(* Logix 5000 project; controller IF2_DEMO Emulate 5570 rev 20.12; software revision 20.04 *)
// RSTechEd 2013 Demo

TASK MainTask (continuous, watchdog 100000 ms) : Main, FillerD, LabelerD
TASK MotionTiming (periodic, rate 25 ms, priority 2, watchdog 50000 ms) : MotionProg

MODULES
   Local : Emulate 5570 (ICP 2, rev 20.12)
END_MODULES

TYPE Controls :   // Workcell Status
STRUCT
   Standby : BOOL;
   StandbyCode : INT;
   Run : BOOL;
   Auto : BOOL;
   Run_sw : BOOL;
END_STRUCT
END_TYPE

TYPE Counts :   // Production Information - Part Counts
STRUCT
   Total : DINT;
   Good : DINT;
   Scrap : DINT;
   BottlesMin : DINT;
END_STRUCT
END_TYPE

TYPE DownTime :   // DownTime Category
STRUCT
   Breakdown : BOOL;
   BreakdownCode : INT;
   UnschedMaint : BOOL;
   Testing : BOOL;
END_STRUCT
END_TYPE

TYPE Event_Triggers :
STRUCT
   EventTrigger : INT;
END_STRUCT
END_TYPE

TYPE Events :
STRUCT
   DownTime : DownTime;
   Operate : Operate;
   Control : Controls;
END_STRUCT
END_TYPE

TYPE FTVPDemoEvents :
STRUCT
   DownTime : DownTime;
   Operate : Operate;
   Control : Controls;
END_STRUCT
END_TYPE

TYPE FTVPDemoLine :
STRUCT
   Downtime : DINT;   // Line Downtime Value
   Runstate : BOOL;   // Running status of the line
   OutputTarget : REAL;   // Target value for production output
   OutputActual : REAL;   // Actual Value of Production Output
   Quality : REAL;   // Line Quality Value
   Rejects : REAL;   // Line Reject Count
END_STRUCT
END_TYPE

TYPE FTVPDemoProduct :
STRUCT
   ProductID : STRING;
   Recipe : STRING;
END_STRUCT
END_TYPE

TYPE FTVPDemoWorkCell :
STRUCT
   LineName : STRING;
   RunState : BOOL;
   Temperature : DINT;
   GoodParts : INT;
   ScrapParts : INT;
   ScrapRate : DINT;
   ProductionRate : DINT;
   Pressure : DINT;
   OrderName : STRING;
   CustomerName : STRING;
   PartName : STRING;
END_STRUCT
END_TYPE

TYPE FTVPSampleMaintenance :
STRUCT
   OperatorLog : STRING;
   MaintenanceActual : DINT;
   MaintenancePlanned : DINT;
   ScheduledDownTime : STRING;
END_STRUCT
END_TYPE

TYPE HMIVars :   // Operator Interface Data
STRUCT
   ScrapRate : REAL;
   SpeedControl : REAL;
   PrevSpeed : REAL;
   CurrentProductionRate : REAL;
   PartCountRollOver : DINT;
   MfgTimeBase : INT;
   MaxEventDur : REAL;
   MinEventDur : REAL;
   EventsPerHr : INT;
   EventDur : REAL;
   RunDur : REAL;
   MinRunDur : REAL;
END_STRUCT
END_TYPE

TYPE IF_OEE :
STRUCT
   Quality : REAL;
   Efficiency : REAL;
   AvailableTime : REAL;
END_STRUCT
END_TYPE

TYPE IPTankLevel :
STRUCT
   Water : Level;
   Chemical : Level;
   Sanitizer : Level;
   RecoveredWater : Level;
END_STRUCT
END_TYPE

TYPE Level :
STRUCT
   Minimum : DINT;
   Maximum : DINT;
   Value : DINT;
END_STRUCT
END_TYPE

TYPE LineData :
STRUCT
   CustomerName : STRING[10];
   PartName : STRING[10];
   OrderName : STRING[10];
   OrderQty : DINT;
END_STRUCT
END_TYPE

TYPE MfgOrders :   // Downloaded Manufacturing Order Details
STRUCT
   CustomerName : STRING;
   OrderName : STRING;
   GetNextOrder : BOOL;
   GetNextOrderStatus : INT;
   OrderQty : DINT;
   OrderQtyStart : DINT;
   ProdRate : REAL;
   SetupTime : REAL;
   PartName : STRING;
   WorkcellName : STRING;
   OperationId : DINT;
   PartNameSav : STRING;
END_STRUCT
END_TYPE

TYPE MLHMI :
STRUCT
   HelpInfo : INT;
   Motor1AmpRate : INT;
   Motor1HighTemp : BOOL;
   Motor1Overload : BOOL;
   Motor2AmpRate : INT;
   Motor2HighTemp : BOOL;
   Motor2Overload : BOOL;
   CustomerName : STRING;
   OEE : INT;
   OrderQTY : INT;
   PartName : STRING;
   ProdRate : INT;
   SetUpTime : INT;
   OrderName : STRING;
END_STRUCT
END_TYPE

TYPE MotionVars :   // Operator Interface Data
STRUCT
   Motion : REAL;
   MotionFactor : REAL;
   MotionMax : REAL;
END_STRUCT
END_TYPE

TYPE OEE :   // Operational Equipment Effectiveness
STRUCT
   IdealCycleTime : REAL;
   Parts : Counts;
END_STRUCT
END_TYPE

TYPE Operate :   // Events related to Operating Workcells
STRUCT
   Setup : BOOL;
   Load : BOOL;
   OrderProc : BOOL;
END_STRUCT
END_TYPE

TYPE PFlex700_Input_I0 :
STRUCT
   DriveStatus : INT;
   DriveStatus_Ready : BOOL;
   DriveStatus_Active : BOOL;
   DriveStatus_CommandDir : BOOL;
   DriveStatus_ActualDir : BOOL;
   DriveStatus_Accelerating : BOOL;
   DriveStatus_Decelerating : BOOL;
   DriveStatus_Alarm : BOOL;
   DriveStatus_Faulted : BOOL;
   DriveStatus_AtSpeed : BOOL;
   DriveStatus_LocalID0 : BOOL;
   DriveStatus_LocalID1 : BOOL;
   DriveStatus_LocalID2 : BOOL;
   DriveStatus_SpdRefID0 : BOOL;
   DriveStatus_SpdRefID1 : BOOL;
   DriveStatus_SpdRefID2 : BOOL;
   DriveStatus_SpdRefID3 : BOOL;
   OutputFreq : INT;
   AccelTime1 : INT;
   DecelTime1 : INT;
   Fault1Code : INT;
   DCBusVoltage : INT;
   OutputCurrent : INT;
   Undefined_C2 : INT;
END_STRUCT
END_TYPE

TYPE PFlex700_Output_O0 :
STRUCT
   DriveLogicRslt : INT;
   DriveLogicRslt_Stop : BOOL;
   DriveLogicRslt_Start : BOOL;
   DriveLogicRslt_Jog : BOOL;
   DriveLogicRslt_ClearFault : BOOL;
   DriveLogicRslt_Forward : BOOL;
   DriveLogicRslt_Reverse : BOOL;
   DriveLogicRslt_LocalContrl : BOOL;
   DriveLogicRslt_MOPInc : BOOL;
   DriveLogicRslt_Accel1 : BOOL;
   DriveLogicRslt_Accel2 : BOOL;
   DriveLogicRslt_Decel1 : BOOL;
   DriveLogicRslt_Decel2 : BOOL;
   DriveLogicRslt_SpdRefID0 : BOOL;
   DriveLogicRslt_SpdRefID1 : BOOL;
   DriveLogicRslt_SpdRefID2 : BOOL;
   DriveLogicRslt_MOPDec : BOOL;
   CommandedFreq : INT;
   AccelTime1 : INT;
   DecelTime1 : INT;
   Undefined_B1 : INT;
   Undefined_B2 : INT;
   Undefined_C1 : INT;
   Undefined_C2 : INT;
END_STRUCT
END_TYPE

TYPE Plant :
STRUCT
   Downtime : REAL;
   Output : REAL;
   Quality : REAL;
END_STRUCT
END_TYPE

TYPE SimVars :   // Variables to Simulated Production
STRUCT
   Cycle : TIMER;
   Run : TIMER;
   Event : TIMER;
   Setup : TIMER;
   Good : REAL;
   Scrap : REAL;
   GoToRun : BOOL;
   GoToEvent : BOOL;
   EventNumber : INT;
   UtilityBool : BOOL[32];
END_STRUCT
END_TYPE

TYPE SodaRecipe :
STRUCT
   Water : DINT;
   Syrup : DINT;
   Acid : DINT;
   CarbonDioxide : DINT;
   Flavor : STRING;
END_STRUCT
END_TYPE

TYPE State :
STRUCT
   LineState : STRING;
END_STRUCT
END_TYPE

TYPE Tank :   // Blending Tanks
STRUCT
   Level : DINT;
   Fill_Valve : STRING;   // 0 = Open, 1 = closed
   Discharge_Valve : STRING;   // 0 = Open, 1 = closed
   CIP_Time : STRING;
   Name : STRING;
END_STRUCT
END_TYPE

TYPE WC :
STRUCT
   EventTrigger : DINT[3];
   EventValue_REAL : REAL[46];
   FlexREAL : REAL[6];
   FlexSTRING : STRING[10];
   IdealCT : REAL;   // Ideal Cycle Time
   TotalParts : REAL;   // Total Parts Produced
   GoodParts : REAL;   // Good Parts Produced
   ScrapParts : REAL;   // Scrap Parts Produced
   EventValueSTRING : STRING[5];
   Shift : REAL;   // Shift Value
   MonitorValue : REAL[25];
   PV : REAL[5];
   FlexINT : INT[6];
END_STRUCT
END_TYPE

TYPE WorkOrder :
STRUCT
   CustomerName : STRING;
   PartName : STRING;
   OrderName : STRING;
   OrderNumber : INT;
   OrderQty : INT;
END_STRUCT
END_TYPE

ADD_ON_INSTRUCTION PFlex_700_AOI   (* revision 1.0 031707 *)
VAR_INPUT
   Cmd_OperOperReq : BOOL;
   Cmd_ProgOperReq : BOOL;
END_VAR
VAR_OUTPUT
   Sts_OperatorModeEnabled : BOOL; {access Read Only, visible}
END_VAR
VAR_INPUT
   Cmd_OperProgReq : BOOL;
   Cmd_ProgProgReq : BOOL;
END_VAR
VAR_OUTPUT
   Sts_ProgramModeEnabled : BOOL; {access Read Only, visible}
   Sts_CommFault : BOOL; {access Read Only, visible}
END_VAR
VAR_INPUT
   Cmd_StartOper : BOOL;
   Cmd_StartProg : BOOL;
   Cmd_StopOper : BOOL;
   Cmd_StopProg : BOOL;
   Cmd_ResetOper : BOOL;
   Cmd_ResetProg : BOOL;
   Cmd_JogOper : BOOL;
   Cmd_JogProg : BOOL;
   Cmd_FwdOper : BOOL;
   Cmd_FwdProg : BOOL;
   Cmd_RevOper : BOOL;
   Cmd_RevProg : BOOL;
   Set_SpeedOper : INT;
   Set_SpeedProg : INT;
   Set_AccelOper : REAL;
   Set_AccelProg : REAL;
   Set_DecelOper : REAL;
   Set_DecelProg : REAL;
   Set_CommFaultTimerPresetOper : DINT := 1000;
   Set_CommFaultTimerPresetProg : DINT := 1000;
   Set_FaceplateAnimation : INT;
END_VAR
VAR_OUTPUT
   Sts_DriveStatus : DINT; {access Read Only}
   Sts_DriveStatus_Ready : BOOL := 1; {access Read Only}
   Sts_DriveStatus_Active : BOOL := 1; {access Read Only}
   Sts_DriveStatus_CommandDir : BOOL; {access Read Only}
   Sts_DriveStatus_ActualDir : BOOL; {access Read Only}
   Sts_DriveStatus_Accelerating : BOOL; {access Read Only}
   Sts_DriveStatus_Decelerating : BOOL; {access Read Only}
   Sts_DriveStatus_Alarm : BOOL; {access Read Only}
   Sts_DriveStatus_Faulted : BOOL; {access Read Only}
   Sts_DriveStatus_AtSpeed : BOOL; {access Read Only}
   Sts_DriveStatus_LocalID0 : BOOL; {access Read Only}
   Sts_DriveStatus_LocalID1 : BOOL; {access Read Only}
   Sts_DriveStatus_LocalID2 : BOOL; {access Read Only}
   Sts_DriveStatus_SpdRefID0 : BOOL; {access Read Only}
   Sts_DriveStatus_SpdRefID1 : BOOL; {access Read Only}
   Sts_DriveStatus_SpdRefID2 : BOOL; {access Read Only}
   Sts_DriveStatus_SpdRefID3 : BOOL; {access Read Only}
   Val_AccelTime1 : REAL; {access Read Only}
   Val_DecelTime1 : REAL; {access Read Only}
   Val_Fault1Code : DINT; {access Read Only}
   Val_DCBusVoltage : DINT; {access Read Only}
END_VAR
VAR_INPUT
   Cmd_LocalContrlProg : BOOL;
   Cmd_MOPIncProg : BOOL;
   Cmd_Accel1Prog : BOOL;
   Cmd_Accel2Prog : BOOL;
   Cmd_Decel1Prog : BOOL;
   Cmd_Decel2Prog : BOOL;
   Cmd_SpdRefID0Prog : BOOL;
   Cmd_SpdRefID1Prog : BOOL;
   Cmd_SpdRefID2Prog : BOOL;
   Cmd_MOPDecProg : BOOL;
   Cmd_LocalContrlOper : BOOL;
   Cmd_MOPIncOper : BOOL;
   Cmd_Accel1Oper : BOOL;
   Cmd_Accel2Oper : BOOL;
   Cmd_Decel1Oper : BOOL;
   Cmd_Decel2Oper : BOOL;
   Cmd_SpdRefID0Oper : BOOL;
   Cmd_SpdRefID1Oper : BOOL;
   Cmd_SpdRefID2Oper : BOOL;
   Cmd_MOPDecOper : BOOL;
   Set_TrendNextPenOper : DINT;
END_VAR
VAR_OUTPUT
   Val_TrendMin : DINT; {access Read Only}
   Val_TrendMax : DINT; {access Read Only}
END_VAR
VAR_INPUT
   Set_CurrentMinOper : DINT;
   Set_CurrentMaxOper : DINT;
   Set_SpeedMinOper : DINT;
   Set_SpeedMaxOper : DINT;
   Set_DCBusVoltageMinOper : DINT;
   Set_DCBusVoltageMaxOper : DINT;
END_VAR
VAR_IN_OUT
   Inp_PowerFlex_700 : PFlex700_Input_I0; {required}
   Out_PowerFlex_700 : PFlex700_Output_O0; {required}
END_VAR
VAR_OUTPUT
   Val_OutputFreq : DINT; {access Read Only}
   Val_OutputCurrent : DINT; {access Read Only}
END_VAR
VAR_INPUT
   Inp_Scaled_Speed_At_32767 : REAL; {required}
   Cmd_OperToProgPermissive : BOOL;
   Cmd_ProgToOperPermissive : BOOL;
END_VAR
VAR
   CommFaultTimer : TIMER := (PRE := 1000);
   CommStatusValue : DINT;
   Set_DeviceNameOper : STRING := 'PF 700';
   Set_SpeedUnitsOper : STRING := 'SPEED';
   OperONS : BOOL;
   SpeedRate : REAL;
END_VAR

ROUTINE Logic   (* ladder *)
// PowerFlex_70_700_AOI
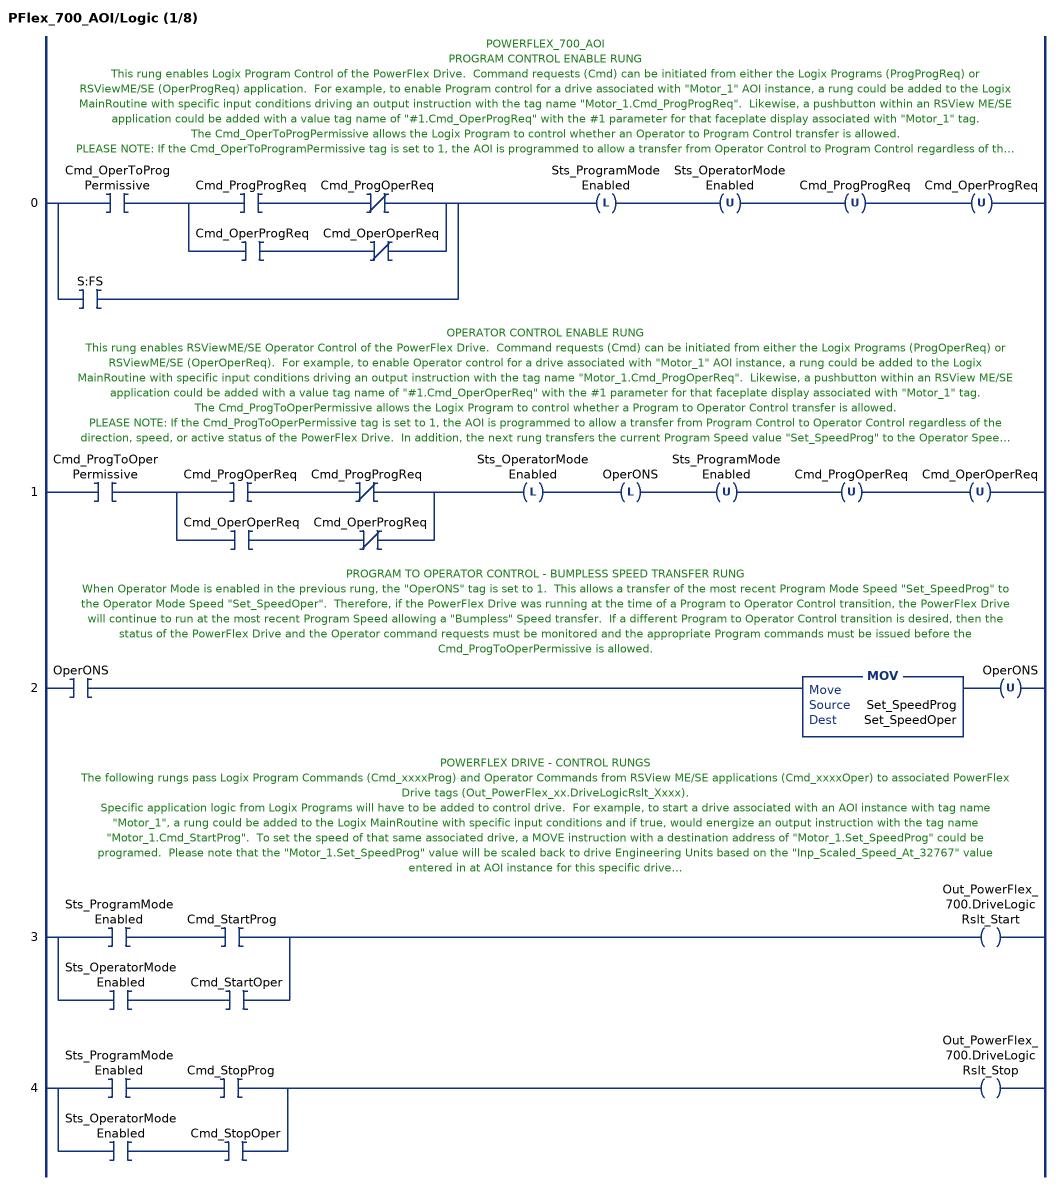
   // POWERFLEX_700_AOI
   // PROGRAM CONTROL ENABLE RUNG
   // This rung enables Logix Program Control of the PowerFlex Drive.  Command requests (Cmd) can be initiated from either the Logix Programs (ProgProgReq) or RSViewME/SE (OperProgReq) application.  For example, to enable Program control for a drive associated with "Motor_1" AOI instance, a rung could be added to the Logix MainRoutine with specific input conditions driving an output instruction with the tag name "Motor_1.Cmd_ProgProgReq".  Likewise, a pushbutton within an RSView ME/SE application could be added with a value tag name of "#1.Cmd_OperProgReq" with the #1 parameter for that faceplate display associated with "Motor_1" tag.
   // The Cmd_OperToProgPermissive allows the Logix Program to control whether an Operator to Program Control transfer is allowed.
   // PLEASE NOTE: If the Cmd_OperToProgramPermissive tag is set to 1, the AOI is programmed to allow a transfer from Operator Control to Program Control regardless of the direction, speed, or active status of the PowerFlex Drive.  Therefore, the status of the PowerFlex Drive must be monitored and used to set Cmd_OperToProgramPermissive tag outside of the AOI to insure a safe transfer.
   0: [XIC(Cmd_OperToProgPermissive) [XIC(Cmd_ProgProgReq) XIO(Cmd_ProgOperReq) ,XIC(Cmd_OperProgReq) XIO(Cmd_OperOperReq) ] ,XIC(S:FS) ]OTL(Sts_ProgramModeEnabled)OTU(Sts_OperatorModeEnabled)OTU(Cmd_ProgProgReq)OTU(Cmd_OperProgReq);
   // OPERATOR CONTROL ENABLE RUNG
   // This rung enables RSViewME/SE Operator Control of the PowerFlex Drive.  Command requests (Cmd) can be initiated from either the Logix Programs (ProgOperReq) or RSViewME/SE (OperOperReq).  For example, to enable Operator control for a drive associated with "Motor_1" AOI instance, a rung could be added to the Logix MainRoutine with specific input conditions driving an output instruction with the tag name "Motor_1.Cmd_ProgOperReq".  Likewise, a pushbutton within an RSView ME/SE application could be added with a value tag name of "#1.Cmd_OperOperReq" with the #1 parameter for that faceplate display associated with "Motor_1" tag.
   // The Cmd_ProgToOperPermissive allows the Logix Program to control whether a Program to Operator Control transfer is allowed.
   // PLEASE NOTE: If the Cmd_ProgToOperPermissive tag is set to 1, the AOI is programmed to allow a transfer from Program Control to Operator Control regardless of the direction, speed, or active status of the PowerFlex Drive.  In addition, the next rung transfers the current Program Speed value "Set_SpeedProg" to the Operator Speed tag, "Set_SpeedOper" tag, creating a "bumpless" transfer when a transfer from Program Control to Operator Control is executed.  Therefore, the status of the PowerFlex Drive must be monitored and appropriate Program commands, for the specific application, must be issued before the Cmd_ProgToOperPermissive tag is set, to insure a safe Program to Operator Control transfer.
   1: XIC(Cmd_ProgToOperPermissive)[XIC(Cmd_ProgOperReq) XIO(Cmd_ProgProgReq) ,XIC(Cmd_OperOperReq) XIO(Cmd_OperProgReq) ]OTL(Sts_OperatorModeEnabled)OTL(OperONS)OTU(Sts_ProgramModeEnabled)OTU(Cmd_ProgOperReq)OTU(Cmd_OperOperReq);
   // PROGRAM TO OPERATOR CONTROL - BUMPLESS SPEED TRANSFER RUNG
   // When Operator Mode is enabled in the previous rung, the "OperONS" tag is set to 1.  This allows a transfer of the most recent Program Mode Speed "Set_SpeedProg" to the Operator Mode Speed "Set_SpeedOper".  Therefore, if the PowerFlex Drive was running at the time of a Program to Operator Control transition, the PowerFlex Drive will continue to run at the most recent Program Speed allowing a "Bumpless" Speed transfer.  If a different Program to Operator Control transition is desired, then the status of the PowerFlex Drive and the Operator command requests must be monitored and the appropriate Program commands must be issued before the Cmd_ProgToOperPermissive is allowed.
   2: XIC(OperONS)MOV(Set_SpeedProg,Set_SpeedOper)OTU(OperONS);
   // POWERFLEX DRIVE - CONTROL RUNGS
   // The following rungs pass Logix Program Commands (Cmd_xxxxProg) and Operator Commands from RSView ME/SE applications (Cmd_xxxxOper) to associated PowerFlex Drive tags (Out_PowerFlex_xx.DriveLogicRslt_Xxxx).
   // Specific application logic from Logix Programs will have to be added to control drive.  For example, to start a drive associated with an AOI instance with tag name "Motor_1", a rung could be added to the Logix MainRoutine with specific input conditions and if true, would energize an output instruction with the tag name "Motor_1.Cmd_StartProg".  To set the speed of that same associated drive, a MOVE instruction with a destination address of "Motor_1.Set_SpeedProg" could be programed.  Please note that the "Motor_1.Set_SpeedProg" value will be scaled back to drive Engineering Units based on the "Inp_Scaled_Speed_At_32767" value entered in at AOI instance for this specific drive.
   // Commands from RSView ME/SE applications will also control the drive when Operator Mode is enabled.  For example, to start a drive associated with "Motor_1" AOI instance, a pushbutton within an RSView ME application with a tag name of "#1.Cmd_StartOper" would have to be configured.  The #1 parameter tagname for that faceplate display would have to be "Motor_1".  To set the speed of that same "Motor_1" associated drive, a numeric input object with the tag name of "#1.Set_SpeedOper" would have to be configured.  Please note that the "#1.Set_SpeedOper" value will be scaled back to drive Engineering Units based on the "Inp_Scaled_Speed_At_32767" value entered in at AOI instance for this specific drive.
   // For ability to set AccelTime1 and DecelTime1, the datalinks within the PowerFlex Drive Module Definitions need to be assigned to these drive parameters.
   3: [XIC(Sts_ProgramModeEnabled) XIC(Cmd_StartProg) ,XIC(Sts_OperatorModeEnabled) XIC(Cmd_StartOper) ]OTE(Out_PowerFlex_700.DriveLogicRslt_Start);
   4: [XIC(Sts_ProgramModeEnabled) XIC(Cmd_StopProg) ,XIC(Sts_OperatorModeEnabled) XIC(Cmd_StopOper) ]OTE(Out_PowerFlex_700.DriveLogicRslt_Stop);
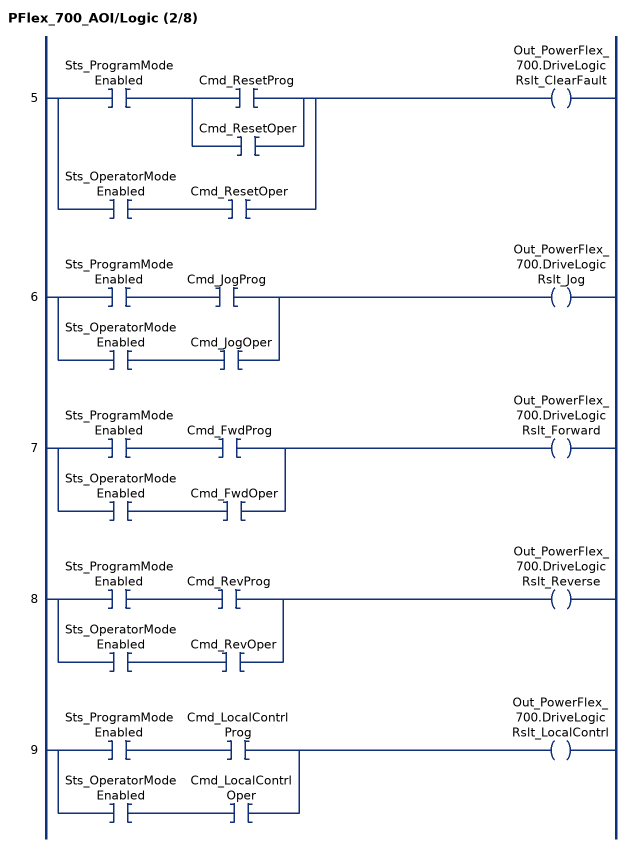
   5: [XIC(Sts_ProgramModeEnabled) [XIC(Cmd_ResetProg) ,XIC(Cmd_ResetOper) ] ,XIC(Sts_OperatorModeEnabled) XIC(Cmd_ResetOper) ]OTE(Out_PowerFlex_700.DriveLogicRslt_ClearFault);
   6: [XIC(Sts_ProgramModeEnabled) XIC(Cmd_JogProg) ,XIC(Sts_OperatorModeEnabled) XIC(Cmd_JogOper) ]OTE(Out_PowerFlex_700.DriveLogicRslt_Jog);
   7: [XIC(Sts_ProgramModeEnabled) XIC(Cmd_FwdProg) ,XIC(Sts_OperatorModeEnabled) XIC(Cmd_FwdOper) ]OTE(Out_PowerFlex_700.DriveLogicRslt_Forward);
   8: [XIC(Sts_ProgramModeEnabled) XIC(Cmd_RevProg) ,XIC(Sts_OperatorModeEnabled) XIC(Cmd_RevOper) ]OTE(Out_PowerFlex_700.DriveLogicRslt_Reverse);
   9: [XIC(Sts_ProgramModeEnabled) XIC(Cmd_LocalContrlProg) ,XIC(Sts_OperatorModeEnabled) XIC(Cmd_LocalContrlOper) ]OTE(Out_PowerFlex_700.DriveLogicRslt_LocalContrl);
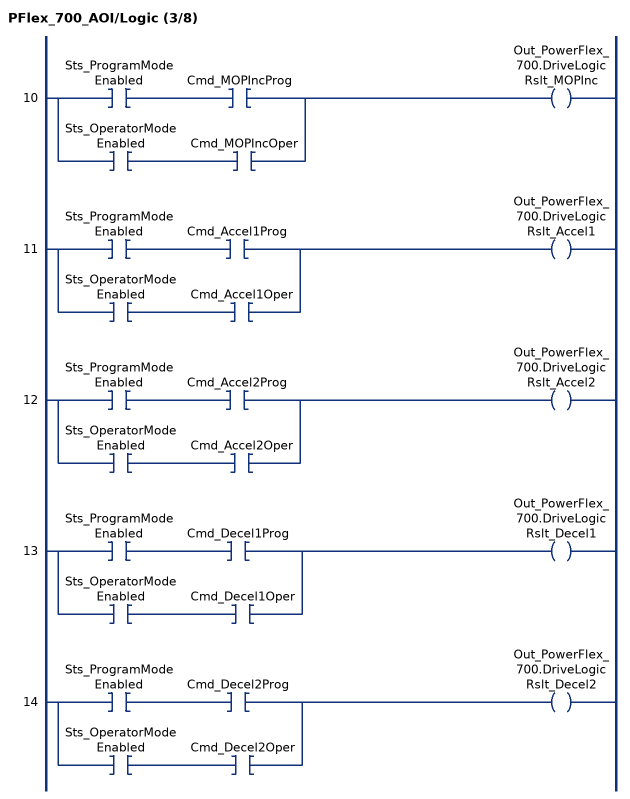
   10: [XIC(Sts_ProgramModeEnabled) XIC(Cmd_MOPIncProg) ,XIC(Sts_OperatorModeEnabled) XIC(Cmd_MOPIncOper) ]OTE(Out_PowerFlex_700.DriveLogicRslt_MOPInc);
   11: [XIC(Sts_ProgramModeEnabled) XIC(Cmd_Accel1Prog) ,XIC(Sts_OperatorModeEnabled) XIC(Cmd_Accel1Oper) ]OTE(Out_PowerFlex_700.DriveLogicRslt_Accel1);
   12: [XIC(Sts_ProgramModeEnabled) XIC(Cmd_Accel2Prog) ,XIC(Sts_OperatorModeEnabled) XIC(Cmd_Accel2Oper) ]OTE(Out_PowerFlex_700.DriveLogicRslt_Accel2);
   13: [XIC(Sts_ProgramModeEnabled) XIC(Cmd_Decel1Prog) ,XIC(Sts_OperatorModeEnabled) XIC(Cmd_Decel1Oper) ]OTE(Out_PowerFlex_700.DriveLogicRslt_Decel1);
   14: [XIC(Sts_ProgramModeEnabled) XIC(Cmd_Decel2Prog) ,XIC(Sts_OperatorModeEnabled) XIC(Cmd_Decel2Oper) ]OTE(Out_PowerFlex_700.DriveLogicRslt_Decel2);
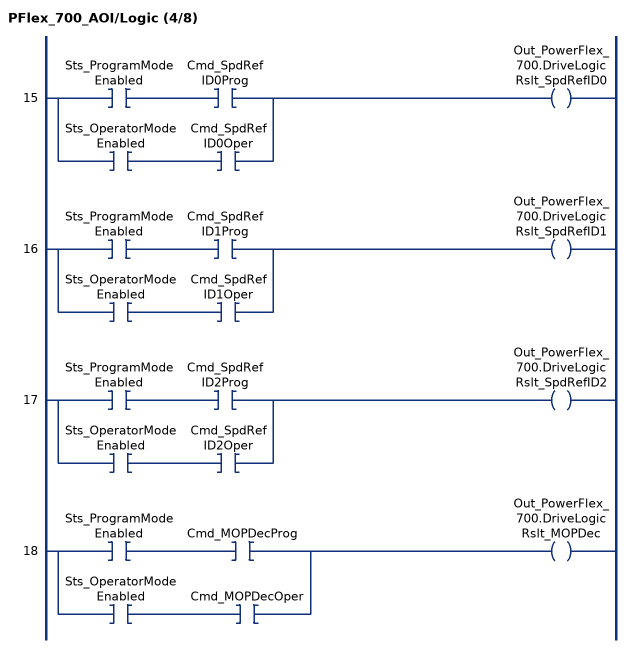
   15: [XIC(Sts_ProgramModeEnabled) XIC(Cmd_SpdRefID0Prog) ,XIC(Sts_OperatorModeEnabled) XIC(Cmd_SpdRefID0Oper) ]OTE(Out_PowerFlex_700.DriveLogicRslt_SpdRefID0);
   16: [XIC(Sts_ProgramModeEnabled) XIC(Cmd_SpdRefID1Prog) ,XIC(Sts_OperatorModeEnabled) XIC(Cmd_SpdRefID1Oper) ]OTE(Out_PowerFlex_700.DriveLogicRslt_SpdRefID1);
   17: [XIC(Sts_ProgramModeEnabled) XIC(Cmd_SpdRefID2Prog) ,XIC(Sts_OperatorModeEnabled) XIC(Cmd_SpdRefID2Oper) ]OTE(Out_PowerFlex_700.DriveLogicRslt_SpdRefID2);
   18: [XIC(Sts_ProgramModeEnabled) XIC(Cmd_MOPDecProg) ,XIC(Sts_OperatorModeEnabled) XIC(Cmd_MOPDecOper) ]OTE(Out_PowerFlex_700.DriveLogicRslt_MOPDec);
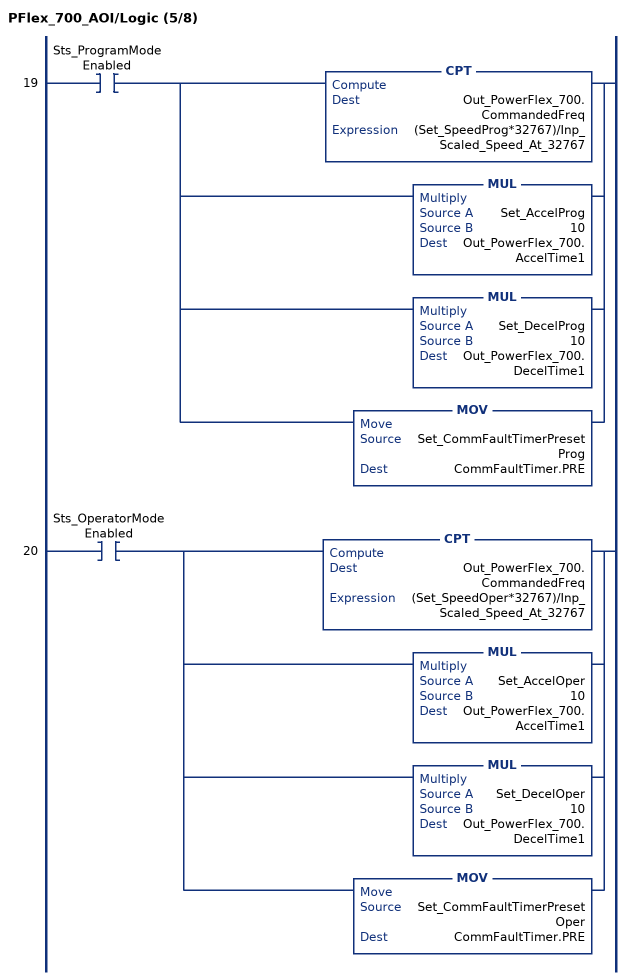
   19: XIC(Sts_ProgramModeEnabled)[CPT(Out_PowerFlex_700.CommandedFreq,(Set_SpeedProg*32767)/Inp_Scaled_Speed_At_32767) ,MUL(Set_AccelProg,10,Out_PowerFlex_700.AccelTime1) ,MUL(Set_DecelProg,10,Out_PowerFlex_700.DecelTime1) ,MOV(Set_CommFaultTimerPresetProg,CommFaultTimer.PRE) ];
   20: XIC(Sts_OperatorModeEnabled)[CPT(Out_PowerFlex_700.CommandedFreq,(Set_SpeedOper*32767)/Inp_Scaled_Speed_At_32767) ,MUL(Set_AccelOper,10,Out_PowerFlex_700.AccelTime1) ,MUL(Set_DecelOper,10,Out_PowerFlex_700.DecelTime1) ,MOV(Set_CommFaultTimerPresetOper,CommFaultTimer.PRE) ];
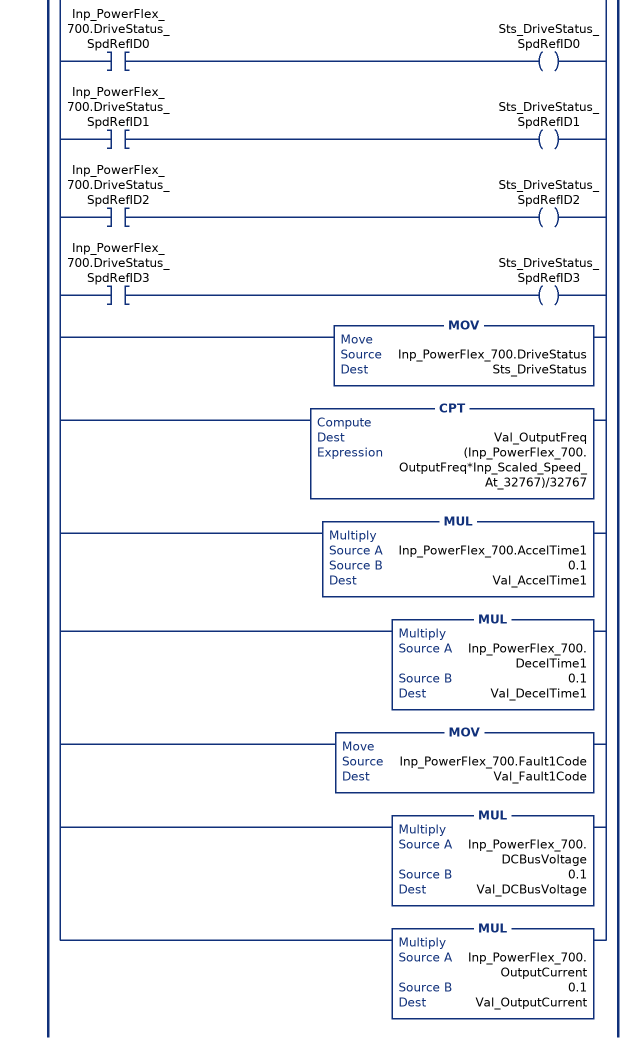
   // POWERFLEX DRIVE - DRIVE STATUS RUNG
   // The following rung simply passes the status information from the associated PowerFlex Drive Status Tags (Inp_PowerFlex_xx.DriveStatus_xxxxx)  to output parameter tags (Sts_DriveStatus_xxxxx) for use by RSView ME/SE applications and Logix Programs.  For example, the "Inp_PowerFlex_xx.DriveStatus_AtSpeed" XIO instruction provides it's status to the AOI status tag "Sts_DriveStatus_AtSpeed".  To provide this "at speed" indication within an RSView ME/SE application for a drive associated with "Motor_1" AOI instance, a multistate indicator could be added with a value tag name of "#1.Sts_DriveStatus_AtSpeed".  The #1 parameter for the faceplate display with the at speed indicator associated with "Motor_1" would be assigned the "Motor_1" tag.  To use this "Sts_DriveStatus_AtSpeed" status for the drive associated with "Motor_1" within a Logix Program routine you would simply assign an input instruction with a tag name of Motor_1.Sts_ DriveStatus_AtSpeed.  Please note that the "Val_OutputFreq" value used by the RSView ME/SE application is scaled based on the "Inp_Scaled_Speed_At_32767" value entered in at AOI instance for the specific drive.
   // In addition, for the ability to display the drive status values and diagnostics, the AccelTime1, DecelTime1, Fault1Code, DCBusVoltage, and OutputCurrent parameter datalinks within the specific PowerFlex Drive Module Definitions need to be configured.
   21: [XIC(Inp_PowerFlex_700.DriveStatus_Ready) OTE(Sts_DriveStatus_Ready) ,XIC(Inp_PowerFlex_700.DriveStatus_Active) OTE(Sts_DriveStatus_Active) ,XIC(Inp_PowerFlex_700.DriveStatus_CommandDir) OTE(Sts_DriveStatus_CommandDir) ,XIC(Inp_PowerFlex_700.DriveStatus_ActualDir) OTE(Sts_DriveStatus_ActualDir) ,XIC(Inp_PowerFlex_700.DriveStatus_Accelerating) OTE(Sts_DriveStatus_Accelerating) ,XIC(Inp_PowerFlex_700.DriveStatus_Decelerating) OTE(Sts_DriveStatus_Decelerating) ,XIC(Inp_PowerFlex_700.DriveStatus_Alarm) OTE(Sts_DriveStatus_Alarm) ,XIC(Inp_PowerFlex_700.DriveStatus_Faulted) OTE(Sts_DriveStatus_Faulted) ,XIC(Inp_PowerFlex_700.DriveStatus_AtSpeed) OTE(Sts_DriveStatus_AtSpeed) ,XIC(Inp_PowerFlex_700.DriveStatus_LocalID0) OTE(Sts_DriveStatus_LocalID0) ,XIC(Inp_PowerFlex_700.DriveStatus_LocalID1) OTE(Sts_DriveStatus_LocalID1) ,XIC(Inp_PowerFlex_700.DriveStatus_LocalID2) OTE(Sts_DriveStatus_LocalID2) ,XIC(Inp_PowerFlex_700.DriveStatus_SpdRefID0) OTE(Sts_DriveStatus_SpdRefID0) ,XIC(Inp_PowerFlex_700.DriveStatus_SpdRefID1) OTE(Sts_DriveStatus_SpdRefID1) ,XIC(Inp_PowerFlex_700.DriveStatus_SpdRefID2) OTE(Sts_DriveStatus_SpdRefID2) ,XIC(Inp_PowerFlex_700.DriveStatus_SpdRefID3) OTE(Sts_DriveStatus_SpdRefID3) ,MOV(Inp_PowerFlex_700.DriveStatus,Sts_DriveStatus) ,CPT(Val_OutputFreq,(Inp_PowerFlex_700.OutputFreq*Inp_Scaled_Speed_At_32767)/32767) ,MUL(Inp_PowerFlex_700.AccelTime1,0.1,Val_AccelTime1) ,MUL(Inp_PowerFlex_700.DecelTime1,0.1,Val_DecelTime1) ,MOV(Inp_PowerFlex_700.Fault1Code,Val_Fault1Code) ,MUL(Inp_PowerFlex_700.DCBusVoltage,0.1,Val_DCBusVoltage) ,MUL(Inp_PowerFlex_700.OutputCurrent,0.1,Val_OutputCurrent) ];
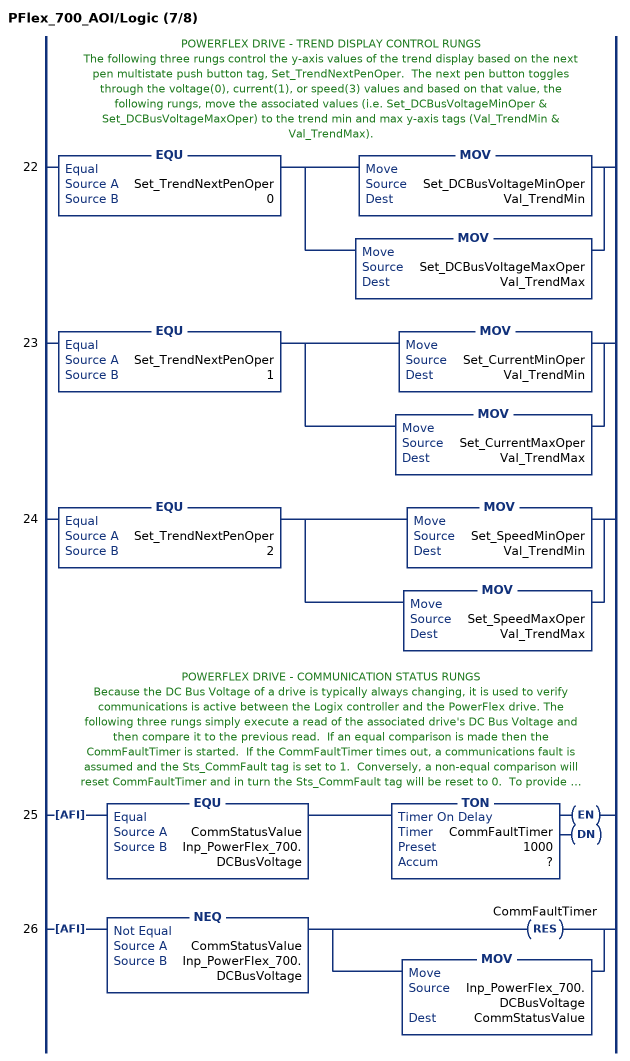
   // POWERFLEX DRIVE - TREND DISPLAY CONTROL RUNGS
   // The following three rungs control the y-axis values of the trend display based on the next pen multistate push button tag, Set_TrendNextPenOper.  The next pen button toggles through the voltage(0), current(1), or speed(3) values and based on that value, the following rungs, move the associated values (i.e. Set_DCBusVoltageMinOper & Set_DCBusVoltageMaxOper) to the trend min and max y-axis tags (Val_TrendMin & Val_TrendMax).
   22: EQU(Set_TrendNextPenOper,0)[MOV(Set_DCBusVoltageMinOper,Val_TrendMin) ,MOV(Set_DCBusVoltageMaxOper,Val_TrendMax) ];
   23: EQU(Set_TrendNextPenOper,1)[MOV(Set_CurrentMinOper,Val_TrendMin) ,MOV(Set_CurrentMaxOper,Val_TrendMax) ];
   24: EQU(Set_TrendNextPenOper,2)[MOV(Set_SpeedMinOper,Val_TrendMin) ,MOV(Set_SpeedMaxOper,Val_TrendMax) ];
   // POWERFLEX DRIVE - COMMUNICATION STATUS RUNGS
   // Because the DC Bus Voltage of a drive is typically always changing, it is used to verify communications is active between the Logix controller and the PowerFlex drive. The following three rungs simply execute a read of the associated drive's DC Bus Voltage and then compare it to the previous read.  If an equal comparison is made then the CommFaultTimer is started.  If the CommFaultTimer times out, a communications fault is assumed and the Sts_CommFault tag is set to 1.  Conversely, a non-equal comparison will reset CommFaultTimer and in turn the Sts_CommFault tag will be reset to 0.  To provide a communication status indication of a drive associated with "Motor_1" AOI instance, an indicator within an RSView ME/SE application with a tag name of "#1.Sts_CommFault" could be added.  The #1 parameter of that associated faceplate display would also need to be assigned to "Motor_1" as well.
   25: AFI()EQU(CommStatusValue,Inp_PowerFlex_700.DCBusVoltage)TON(CommFaultTimer,?,?);
   26: AFI()NEQ(CommStatusValue,Inp_PowerFlex_700.DCBusVoltage)[RES(CommFaultTimer) ,MOV(Inp_PowerFlex_700.DCBusVoltage,CommStatusValue) ];
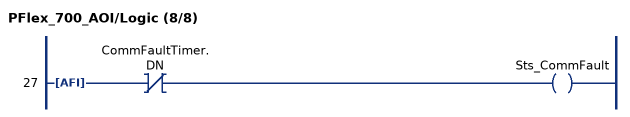
   27: AFI()XIO(CommFaultTimer.DN)OTE(Sts_CommFault);
END_ROUTINE
END_ADD_ON_INSTRUCTION

VAR_GLOBAL   (* controller tags *)
   AlarmFillerConvJam : BOOL;
   AlarmLabelJam : BOOL;
   AlarmMotorOverHeat : BOOL := 1;
   AlarmPaperOut : BOOL;
   AlarmTank1DiscJam : BOOL;
   AlarmTank1Jam_Ack : BOOL := 1;
   AlarmTank2DiscJam : BOOL;
   AlarmTank2FillJam : BOOL;
   AlarmTank2Jam_Shelve : BOOL;
   AlarmTank2Jam_ShelveTime : DINT := 2;
   BlueBerry : FTVPDemoProduct := (ProductID := 'BLB', Recipe := 'BLB038RCP');
   Cases_Rejects_Line1 : DINT;
   ChangeOver_In_Progress : BOOL;
   ChemConc : DINT := 22;
   chemValveFlow : DINT;
   CIP_String_Creator : STRING := '/';
   CIP_TimeStamp : STRING := '2014/4/2';
   CIP_TimeStamp_Day : STRING := '2';
   CIP_TimeStamp_Month : STRING := '4';
   CIP_TimeStamp_Year : STRING;
   CIPActive : BOOL := 1;
   CIPAlarm_Start : BOOL := 1;
   CIPAlarmTrigger : BOOL[32] := ([0] := 1, [1] := 1, [2] := 1, [3] := 1);
   CIPClarity : DINT := 99;
   CIPCounter : COUNTER[4] := ([0].PRE := 20000, [1].PRE := 20000, [2].PRE := 20000, [3].PRE := 20000, [3].ACC := -2, [3].CD := 1);
   CIPFilling : BOOL[32];
   CIPTankColour : DINT[4] := ([1] := 1, [2] := 2, [3] := 3);
   CIPTestCounter : COUNTER;
   CIPTimer : TIMER[4] := ([0].PRE := 7500, [0].ACC := 7500, [0].EN := 1, [0].DN := 1, [1].PRE := 1500, [1].EN := 1, [1].DN := 1, [2].PRE := 6000, [2].ACC := 6000, [2].EN := 1, [2].DN := 1, [3].PRE := 6000, [3].ACC := 6000, [3].EN := 1, [3].DN := 1);
   CIPValve0 : ALARM_DIGITAL;
   CIPValve1 : ALARM_DIGITAL;
   CIPValve2 : ALARM_DIGITAL;
   CIPValve3 : ALARM_DIGITAL;
   Current_Order : STRING := 'GF-08-CZ-525';
   CurrentCustomerName : STRING := 'Soda Inc.';
   CurrentPartName : STRING := 'GF-11';
   Delay : TIMER[4] := ([0].PRE := 500, [0].ACC := 500, [0].EN := 1, [0].DN := 1, [1].PRE := 50, [1].ACC := 50, [1].EN := 1, [1].DN := 1, [2].PRE := 500, [2].ACC := 500, [2].EN := 1, [2].DN := 1, [3].PRE := 500, [3].ACC := 500, [3].EN := 1, [3].DN := 1);
   Delay2 : TIMER := (PRE := 5000);
   DispenserLine : LineData := (CustomerName[0] := 'Big-Mart', CustomerName[1] := 'Soda Inc.', CustomerName[2] := 'Pop World', CustomerName[3] := 'Soda Co.', PartName[0] := 'BL-22', PartName[1] := 'GF-11', PartName[2] := 'MG98', PartName[3] := 'KW02', OrderName[0] := 'WO-02-AD');
   Filler_Bottles_Per_Minute : ALIAS FOR ProdCounts.Total;
   Filler_Stopped : BOOL;
   Filling : BOOL;
   Grapefruit : FTVPDemoProduct := (ProductID := 'GPF', Recipe := 'GPF022RCP');
   HMI_Motion : COUNTER := (PRE := 100, ACC := 94, CU := 1);
   HMISystemClock : DINT[7] := ([0] := 2012, [1] := 4, [2] := 24, [3] := 23, [4] := 25, [5] := 25);
   IF_OEE : IF_OEE := (Quality := 0.8855981, Efficiency := 0.7758806, AvailableTime := 0.91280067);
   InitializeDelay : TIMER := (PRE := 4000);
   InstantFizz_Plant : Plant := (Downtime := 5.0, Output := 1.557223, Quality := 0.8869268);
   Kiwi : FTVPDemoProduct := (ProductID := 'KWI', Recipe := 'KWI002RCP');
   Labeler_Stopped : BOOL;
   LastOrderCount : DINT := 48;
   LastOrderNumber : STRING := 'GF-08-CZ-525';
   Line1 : FTVPDemoLine := (Runstate := 1, OutputTarget := 1.5, OutputActual := 1.5644453, Quality := 0.8855981, Rejects := 0.15644453);
   Line_State_String : State := (LineState := 'Running');
   LineStates : STRING[4] := ([0] := 'Stopped', [1] := 'Running', [2] := 'Starved', [3] := 'Blocked');
   Mango : FTVPDemoProduct := (ProductID := 'MGO', Recipe := 'MGO003RCP');
   ManualCompleted : BOOL;
   Menu_GOTO_dx : DINT := 10;
   Menu_GOTO_H : DINT := 461;
   Menu_GOTO_POS : DINT := 470;
   MixAgitatorDelayTimer : TIMER := (PRE := 5000);
   MIXCIPStep_DelayTimer : TIMER := (PRE := 10000);
   MixSteps : DINT := 7;   // 1=Initializing 2=Adding Water 3=Wait for manual 4=Agitate 5=xfer 6=cip 7=complete
   MixTransferOutTimer : TIMER := (PRE := 10000);
   MLHMI : MLHMI := (HelpInfo := 99, Motor1AmpRate := 80, Motor2AmpRate := 95, OrderQTY := 6, ProdRate := 5);
   MotionSimClr : DINT;
   MotionSimCntr : COUNTER[10] := ([0].PRE := 200, [0].ACC := 93, [1].PRE := 200, [1].ACC := 17);
   MotionSimCount : DINT[10] := ([0] := 17, [1] := 1);
   MotionSimEn : DINT;
   Motor_1 : PFlex_700_AOI := (Sts_ProgramModeEnabled := 1, Set_CommFaultTimerPresetOper := 1000, Set_CommFaultTimerPresetProg := 1000, Inp_Scaled_Speed_At_32767 := 1000.0, Cmd_OperToProgPermissive := 1, Cmd_ProgToOperPermissive := 1);
   Motor_1_I : PFlex700_Input_I0;
   Motor_1_I1 : PFlex700_Output_O0;
   MotorOverheatAlarm : ALARM_ANALOG;
   MotorTemp : DINT := 1001;
   NewOrder_Trigger : Event_Triggers := (EventTrigger := 100);
   Next_Order : STRING := 'MG-01-RZ-970';
   Next_Product : DINT := 1;
   OEE_Part_Scrap_Old : DINT;
   OEE_Parts_Good_Old : DINT;
   OEE_Parts_Total_Old : DINT;
   OEE_Scrap_Filler : DINT := 26;
   OEE_Scrap_Labeler : DINT := 185;
   OEE_Scrap_Packaging : DINT := 75;
   OrderQty : DINT[4] := ([0] := 3600);
   Packaging_Stopped : BOOL;
   PartCountRollOver : DINT;
   Performance_Control : DINT := 2;
   Phase_1 : PHASE := (State := 64, Idle := 1);
   Phase_2 : PHASE := (State := 64, Idle := 1);
   Phase_Timer : TIMER := (PRE := 15000, ACC := 229, EN := 1, TT := 1);
   Previous_Order : STRING := 'BL-03-RM-662';
   PreviousCustomerName : STRING := 'Big-Mart';
   PreviousPartName : STRING := 'BL-22';
   ProdCounts : Counts := (Total := 1590, Good := 1403, Scrap := 187, BottlesMin := 119);
   Product_Change : DINT;
   Production_Start_Labeler : BOOL := 1;
   Production_Start_Packaging : BOOL := 1;
   ProductionStart : BOOL := 1;
   ProductionStop : BOOL;
   RapidMixActive : BOOL;
   RapidMixTimer : TIMER := (PRE := 10000);
   RefillLine : LineData := (CustomerName[0] := 'Big-Mart', PartName[0] := 'Apple-R40', OrderName[0] := 'WO-44-SR', OrderQty := 30000);
   RotateTimer : TIMER := (PRE := 10000, ACC := 3523, EN := 1, TT := 1);
   Run_Day : INT := 171;
   Run_Hr : INT := 5;
   Run_Min : INT := 6;
   Run_Sec : INT := 46;
   Run_Timer : TIMER := (PRE := 1000, ACC := 708, EN := 1, TT := 1);
   SanConc : DINT := 39;
   Snapshot : STRING := 'snapshot';
   SodaCIPTanks : IPTankLevel := (Water.Maximum := 20000, Water.Value := 1500, Chemical.Minimum := 1000, Chemical.Maximum := 8000, Chemical.Value := 6000, Sanitizer.Minimum := 2000, Sanitizer.Maximum := 10000, Sanitizer.Value := 6000, RecoveredWater.Minimum := 5000, RecoveredWater.Maximum := 15000, RecoveredWater.Value := 7500);
   Starve_Block_Filler_Start_Toggle : BOOL;
   Starve_Block_Labeler_Start_Toggle : BOOL;
   Starve_Block_Packaging_Start_Toggle : BOOL;
   Step2 : BOOL;
   T1 : BOOL;
   T2 : BOOL;
   TankValue : DINT[4] := ([0] := 12500, [1] := 20000, [2] := 1982, [3] := 2000);
   TempCalc3 : DINT[4] := ([3] := 40012);
   testAlarm : BOOL;
   Timer1000ms : TIMER := (PRE := 1000, ACC := 544, EN := 1, TT := 1);
   Timer100ms : TIMER := (PRE := 100, ACC := 34, EN := 1, TT := 1);
   Timer10ms : TIMER := (PRE := 10, ACC := 10, EN := 1, DN := 1);
   Timer1ms : TIMER := (PRE := 1, EN := 1, TT := 1);
   Timer250ms : TIMER := (PRE := 250, ACC := 55, EN := 1, TT := 1);
   Timer500ms : TIMER := (PRE := 500, ACC := 458, EN := 1, TT := 1);
   TimeTrigger : BOOL;
   Valve : STRING[4] := ([0] := 'Recovered Water', [1] := 'Water Valve', [2] := 'Chemicals Valve', [3] := 'Sanitizer Valve');
   ValveFlowOn : BOOL := 1;
   WallClock : DINT[7] := ([0] := 2014, [1] := 4, [2] := 2, [3] := 19, [4] := 33, [5] := 44, [6] := 856004);
   WaterLevelDefault : DINT := 14000;
   WC : WC[10] := ([0].EventTrigger[0] := 258, [0].EventValue_REAL[1] := 3.0, [0].EventValue_REAL[2] := 4.0, [0].FlexSTRING[0] := 'BL-22', [0].FlexSTRING[3] := 'WO-02-AD', [0].FlexSTRING[4] := 'Big-Mart', [0].IdealCT := 2.0, [0].TotalParts := 2615.9812, [0].GoodParts := 2589.8208, [0].ScrapParts := 26.160408, [0].MonitorValue[0] := 1.0, [0].PV[0] := 172.14752, [0].PV[1] := 155.1654, [1].EventValue_REAL[2] := 5.0, [1].FlexREAL[1] := 3.0, [1].FlexSTRING[0] := 'Apple-R40', [1].FlexSTRING[3] := 'WO-44-SR', [1].FlexSTRING[4] := 'Big-Mart', [1].IdealCT := 3.0, [1].MonitorValue[0] := 1.0, [1].MonitorValue[1] := 1.0, [1].PV[0] := 179.6136, [1].PV[1] := 155.00154, [2].EventTrigger[0] := 256, [2].EventValue_REAL[1] := 3.0, [2].EventValue_REAL[2] := 2.0, [2].FlexSTRING[0] := 'BL-22', [2].FlexSTRING[3] := 'WO-02-AD', [2].FlexSTRING[4] := 'Big-Mart', [2].IdealCT := 2.0, [2].MonitorValue[0] := 2.0, [2].MonitorValue[2] := 2.0, [2].PV[0] := 147.97226, [2].PV[1] := 165.06796, [3].EventValue_REAL[1] := 3.0, [3].EventValue_REAL[2] := 1.0, [3].FlexSTRING[0] := 'Apple-R40', [3].FlexSTRING[3] := 'WO-44-SR', [3].FlexSTRING[4] := 'Big-Mart', [3].IdealCT := 3.0, [3].MonitorValue[0] := 2.0, [3].MonitorValue[3] := 1.0, [3].PV[0] := 206.22862, [3].PV[1] := 186.84538, [4].EventTrigger[0] := 258, [4].EventValue_REAL[1] := 6.0, [4].EventValue_REAL[2] := 4.0, [4].FlexSTRING[0] := 'BL-22', [4].FlexSTRING[3] := 'WO-02-AD', [4].FlexSTRING[4] := 'Big-Mart', [4].IdealCT := 2.0, [4].TotalParts := 1589.555, [4].GoodParts := 1403.0316, [4].ScrapParts := 186.5234, [4].MonitorValue[0] := 2.0, [4].MonitorValue[4] := 2.0, [4].PV[0] := 163.94368, [4].PV[1] := 144.1438, [5].EventValue_REAL[1] := 3.0, [5].EventValue_REAL[2] := 4.0,
        [5].FlexSTRING[0] := 'Apple-R40', [5].FlexSTRING[3] := 'WO-44-SR', [5].FlexSTRING[4] := 'Big-Mart', [5].IdealCT := 4.0, [5].MonitorValue[0] := 2.0, [5].MonitorValue[5] := 1.0, [5].PV[0] := 200.60545, [5].PV[1] := 168.83234, [6].EventTrigger[0] := 2048, [6].EventValue_REAL[1] := 3.0, [6].IdealCT := 5.0, [7].EventTrigger[0] := 2048, [7].EventValue_REAL[1] := 3.0, [7].IdealCT := 5.0, [8].EventTrigger[0] := 2, [8].EventValue_REAL[1] := 3.0, [8].EventValue_REAL[2] := 4.0, [8].FlexSTRING[0] := 'BL-22', [8].FlexSTRING[3] := 'WO-02-AD', [8].FlexSTRING[4] := 'Big-Mart', [8].IdealCT := 2.0, [8].TotalParts := 2501.9592, [8].GoodParts := 2426.899, [8].ScrapParts := 75.06019, [8].MonitorValue[0] := 2.0, [8].MonitorValue[8] := 2.0, [8].PV[0] := 172.14752, [8].PV[1] := 155.1654, [9].EventValue_REAL[1] := 3.0, [9].EventValue_REAL[2] := 4.0, [9].FlexSTRING[0] := 'Apple-R40', [9].FlexSTRING[3] := 'WO-44-SR', [9].FlexSTRING[4] := 'Big-Mart', [9].IdealCT := 2.0, [9].MonitorValue[9] := 2.0, [9].PV[0] := 219.43391, [9].PV[1] := 197.2076);
   WorkOrder : WorkOrder := (CustomerName := 'Soda Inc.', PartName := 'GF-11', OrderName := 'GF-08-CZ-525', OrderNumber := 525, OrderQty := 3600);
END_VAR

PROGRAM Blending   (* main routine Agitator *)
// TechEd 2008 Soda Demo
VAR
   Agitator : DISCRETE_2STATE := (ProgCommand := 1, State0Perm := 1, State1Perm := 1, FB1 := 1, Out := 1, CommandStatus := 1);
   CIP_TimeStamp : STRING;
   GRT_01 : FBD_COMPARE := (SourceA := 100.0, SourceB := 20.0, Dest := 1);
   Recipe : SodaRecipe := (Water := 200, Syrup := 50, Acid := 4, CarbonDioxide := 2, Flavor := 'Mango');
   SodaDate : STRING[7] := ([0] := '2008', [1] := '5', [2] := '7', [3] := '18', [4] := '4', [5] := '2', [6] := '2008\5\7  ');
   SodaMonth : STRING;
   SodaSpace : STRING := '  ';
   SodaYear : STRING := '\';
   Tank1 : Tank := (Level := 400, Fill_Valve := 'Open', Discharge_Valve := 'Open', CIP_Time := '2011/6/13', Name := 'Tank1');
   Tank2 : Tank := (Level := 250, Fill_Valve := 'Open', Discharge_Valve := 'Closed', CIP_Time := '2011/6/13', Name := 'Tank2');
   Tank3 : Tank := (Fill_Valve := 'Closed', Discharge_Valve := 'Closed', CIP_Time := '2011/6/13', Name := 'Tank3');
   TankAlm : TIMER := (PRE := 360000, ACC := 51270);
   TankLevel : DINT := 100;
   TONR_01 : FBD_TIMER := (TimerEnable := 1, ACC := 10, EN := 1, DN := 1);
END_VAR

ROUTINE Agitator   (* function block diagram *)
   SHEET 1
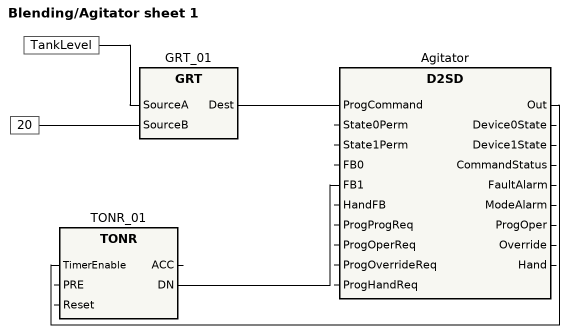
   TONR_01 : TONR(TimerEnable := Agitator.Out {feedback});   // unwired pins: PRE Reset ACC
   GRT_01 : GRT(SourceA := TankLevel, SourceB := 20);
   Agitator : D2SD(ProgCommand := GRT_01.Dest {feedback}, FB1 := TONR_01.DN);   // unwired pins: State0Perm State1Perm FB0 HandFB ProgProgReq ProgOperReq ProgOverrideReq ProgHandReq Device0State Device1State CommandStatus FaultAlarm ModeAlarm ProgOper Override Hand
END_ROUTINE

ROUTINE MainRoutine   (* ladder *)
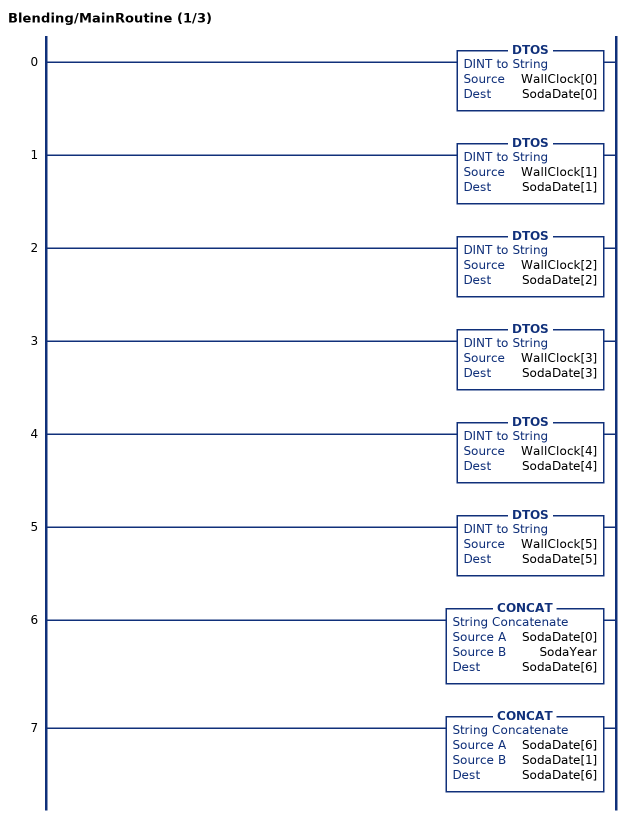
   0: DTOS(WallClock[0],SodaDate[0]);
   1: DTOS(WallClock[1],SodaDate[1]);
   2: DTOS(WallClock[2],SodaDate[2]);
   3: DTOS(WallClock[3],SodaDate[3]);
   4: DTOS(WallClock[4],SodaDate[4]);
   5: DTOS(WallClock[5],SodaDate[5]);
   6: CONCAT(SodaDate[0],SodaYear,SodaDate[6]);
   7: CONCAT(SodaDate[6],SodaDate[1],SodaDate[6]);
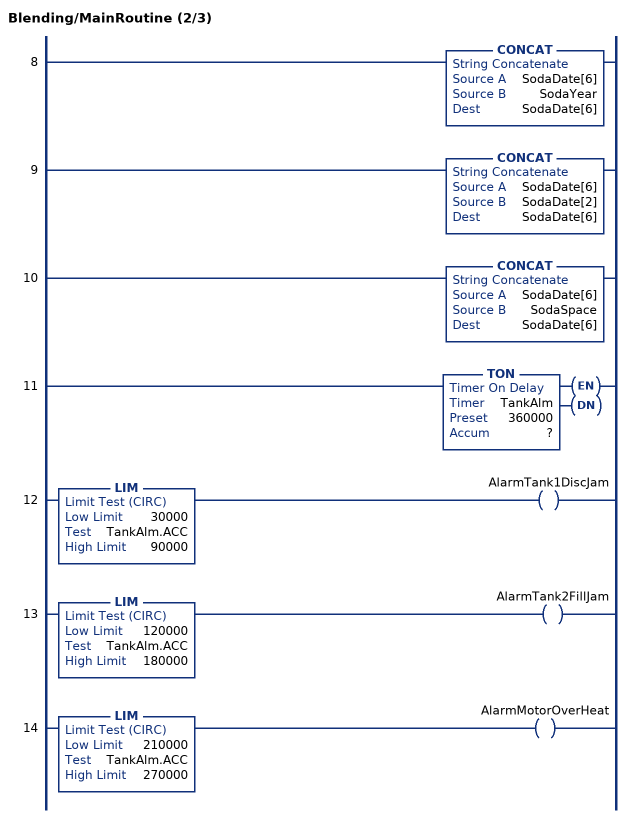
   8: CONCAT(SodaDate[6],SodaYear,SodaDate[6]);
   9: CONCAT(SodaDate[6],SodaDate[2],SodaDate[6]);
   10: CONCAT(SodaDate[6],SodaSpace,SodaDate[6]);
   11: TON(TankAlm,?,?);
   12: LIM(30000,TankAlm.ACC,90000)OTE(AlarmTank1DiscJam);
   13: LIM(120000,TankAlm.ACC,180000)OTE(AlarmTank2FillJam);
   14: LIM(210000,TankAlm.ACC,270000)OTE(AlarmMotorOverHeat);
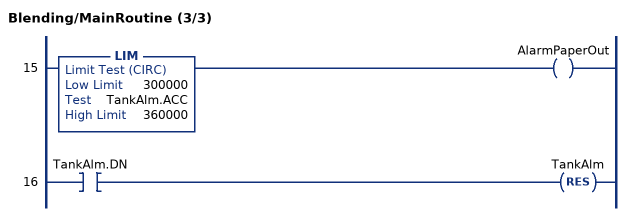
   15: LIM(300000,TankAlm.ACC,360000)OTE(AlarmPaperOut);
   16: XIC(TankAlm.DN)RES(TankAlm);
END_ROUTINE
END_PROGRAM

PROGRAM CapperD
VAR
   BadBoxes : INT := -11247;
   Block_Delay : TIMER := (PRE := 15000);
   Blocked_L : BOOL;
   BottleCount : DINT := 132;
   BottleCounter : COUNTER := (PRE := 50000, ACC := 9);
   BottleMotion1 : TIMER := (PRE := 480, ACC := 180, EN := 1, TT := 1);
   BottlesVSCases : BOOL := 1;
   CaseCount : DINT := 3600;
   CaseCounter : COUNTER := (PRE := 50000, ACC := 2, CU := 1);
   CaseLineSpeed : DINT := 950;
   CaseLineSpeedTemp : DINT := 950;
   CaseMotion1 : TIMER := (PRE := 1050);
   CasesVSBottles : BOOL;
   ControlPanelCount : COUNTER := (DN := 1);
   ControlPanelDone : BOOL;
   ControlPanelDown : BOOL;
   ControlPanelSpeed : TIMER := (PRE := 50, ACC := 22, EN := 1, TT := 1);
   Ctrl_Bit : BOOL;
   Divisor1 : DINT := 12;
   Divisor2 : DINT := 21;
   DownStream_Run : ALIAS FOR WC[4].EventTrigger[0].1;
   DownStream_Running : ALIAS FOR WC[4].EventTrigger[0].8;
   Events : Events := (DownTime.BreakdownCode := 2, DownTime.UnschedMaint := 1, Control.StandbyCode := 1, Control.Auto := 1);
   Events_Control_Auto : ALIAS FOR WC_L.EventTrigger[0].5;
   Events_Control_OpStop : ALIAS FOR WC_L.EventTrigger[0].3;
   Events_Control_Run : ALIAS FOR WC_L.EventTrigger[0].1;
   Events_Control_Running : ALIAS FOR WC_L.EventTrigger[0].8;
   Events_Control_Standby : ALIAS FOR WC_L.EventTrigger[0].0;
   Events_Control_StandbyCode : ALIAS FOR WC_L.EventValue_REAL[1];
   Events_DownTime_Breakdown : ALIAS FOR WC_L.EventTrigger[0].2;
   Events_DownTime_BreakdownCode : ALIAS FOR WC_L.EventValue_REAL[2];
   Events_DownTime_Testing : ALIAS FOR WC_L.EventTrigger[0].7;
   Events_DownTime_UnschedMaint : ALIAS FOR WC_L.EventTrigger[0].6;
   Events_Operate_Load : ALIAS FOR WC_L.EventTrigger[0].10;
   Events_Operate_OrderProc : ALIAS FOR WC_L.EventTrigger[0].11;
   Events_Operate_Setup : ALIAS FOR WC_L.EventTrigger[0].9;
   HighBottleSpeed : BOOL;
   HMI : HMIVars := (ScrapRate := 5.0, SpeedControl := 90.0, PrevSpeed := 100.0, PartCountRollOver := 9999999, MfgTimeBase := 1, MaxEventDur := 22.0, MinEventDur := 9.0, EventsPerHr := 100, EventDur := 21.705135, RunDur := 13.938431, MinRunDur := 5.0);
   Math1 : DINT := 1320;
   Math2 : DINT := 1800;
   MaxPsiSP_Capper : DINT := 100;
   MaxPsiSP_Filler : DINT := 120;
   MfgOrders : MfgOrders := (CustomerName := 'Big-Mart', OrderName := 'A123', OrderQty := 40000, ProdRate := 60.0, PartName := 'Apple-D12', WorkcellName := 'CapperD', OperationId := 3, PartNameSav := 'Apple-D12');
   MfgOrders_CustomerName : ALIAS FOR WC_L.FlexSTRING[4];
   MfgOrders_OrderName : ALIAS FOR WC_L.FlexSTRING[3];
   MfgOrders_PartName : ALIAS FOR WC_L.FlexSTRING[0];
   MinPsiSP_Capper : DINT;
   MinPsiSP_Filler : DINT := 5;
   Motion : DINT := 18;
   Motion1Bit : BOOL := 1;
   Motion2Bit : BOOL := 1;
   Motion_Counter : DINT := 1;
   Motion_Speed : DINT := 13;
   Motion_Speed_Divisor : DINT := 4;
   MotionCount : TIMER := (PRE := 1170);
   MotionHolder1 : DINT := 15;
   MotionHolder2 : DINT := 50;
   OEE : OEE := (IdealCycleTime := 2.0);
   OEE_IdealCycleTime : ALIAS FOR WC_L.IdealCT;
   OEE_Parts_Good : ALIAS FOR WC_L.GoodParts;
   OEE_Parts_Scrap : ALIAS FOR WC_L.ScrapParts;
   OEE_Parts_Total : ALIAS FOR WC_L.TotalParts;
   onsbits : DINT;
   OperatorID : ALIAS FOR WC_L.FlexREAL[1];
   Pressure1 : ALIAS FOR WC_L.PV[0];   // PSI
   Pressure_Capper : DINT := 79;
   Pressure_Filler : DINT := 99;
   Pressure_Monitor_ON : BOOL := 1;
   Pressure_rate : REAL := 1.e-04;
   ProductColorCode : INT;
   Reset1Bit : BOOL;
   SecondTimer1 : TIMER := (PRE := 5000, ACC := 4165, EN := 1, TT := 1);
   SecondTimer2 : TIMER := (PRE := 5000, ACC := 1062, EN := 1, TT := 1);
   SecondTimer3 : TIMER := (PRE := 60000, ACC := 1500, EN := 1, TT := 1);
   SIM : SimVars := (Run.PRE := 13938, Event.PRE := 9000, Setup.PRE := 9000, EventNumber := 10, UtilityBool[2] := 1);
        .UTILITYBOOL[2]   // First Scan Bit
   Sin_input_float : REAL := 0.70940536;
   Starve_Delay : TIMER := (PRE := 15000);
   Starved_L : BOOL;
   StateValue : ALIAS FOR WC[2].MonitorValue[0];
   StatusPanelCount : COUNTER := (ACC := 11, DN := 1);
   StatusPanelDone : BOOL := 1;
   StatusPanelDown : BOOL := 1;
   Suppress : Events;
   Temperature1 : ALIAS FOR WC_L.PV[1];   // DEG
   TotalBottleCount : DINT := 1320;
   UpStream_Run : ALIAS FOR WC[0].EventTrigger[0].1;
   UpStream_Running : ALIAS FOR WC[0].EventTrigger[0].8;
   WC_L : ALIAS FOR WC[2];
END_VAR
END_PROGRAM

PROGRAM CapperR   (* main routine MainRoutine *)
VAR
   Block_Delay : TIMER := (PRE := 15000);
   Blocked_L : BOOL;
   Blocked_L1 : BOOL;
   BottleCount : DINT := 298;
   BottleCounter : COUNTER := (PRE := 50000, ACC := 43);
   BottleMotion1 : TIMER := (PRE := 200, ACC := 93, EN := 1, TT := 1);
   Ctrl_Bit : BOOL := 1;
   Divisor1 : DINT := 5;
   DownStream_Run : ALIAS FOR WC[5].EventTrigger[0].1;
   DownStream_Running : ALIAS FOR WC[5].EventTrigger[0].8;
   Events : Events := (DownTime.BreakdownCode := 5, Control.StandbyCode := 1, Control.Run := 1, Control.Auto := 1);
   Events_Control_Auto : ALIAS FOR WC_L.EventTrigger[0].5;
   Events_Control_OpStop : ALIAS FOR WC_L.EventTrigger[0].3;
   Events_Control_Run : ALIAS FOR WC_L.EventTrigger[0].1;
   Events_Control_Running : ALIAS FOR WC_L.EventTrigger[0].8;
   Events_Control_Standby : ALIAS FOR WC_L.EventTrigger[0].0;
   Events_Control_StandbyCode : ALIAS FOR WC_L.EventValue_REAL[1];
   Events_DownTime_Breakdown : ALIAS FOR WC_L.EventTrigger[0].2;
   Events_DownTime_BreakdownCode : ALIAS FOR WC_L.EventValue_REAL[2];
   Events_DownTime_Testing : ALIAS FOR WC_L.EventTrigger[0].7;
   Events_DownTime_UnschedMaint : ALIAS FOR WC_L.EventTrigger[0].6;
   Events_Operate_Load : ALIAS FOR WC_L.EventTrigger[0].10;
   Events_Operate_OrderProc : ALIAS FOR WC_L.EventTrigger[0].11;
   Events_Operate_Setup : ALIAS FOR WC_L.EventTrigger[0].9;
   HMI : HMIVars := (ScrapRate := 5.0, SpeedControl := 100.0, PrevSpeed := 100.0, PartCountRollOver := 9999999, MfgTimeBase := 1, MaxEventDur := 11.0, MinEventDur := 4.0, EventsPerHr := 50, EventDur := 10.953963, RunDur := 59.63427, MinRunDur := 5.0);
   MfgOrders : MfgOrders := (CustomerName := 'Big-Mart', OrderName := 'BB21', OrderQty := 30000, ProdRate := 60.0, PartName := 'STRAW-R40', WorkcellName := 'CapperR', PartNameSav := 'STRAW-R40');
   MfgOrders_CustomerName : ALIAS FOR WC_L.FlexSTRING[4];
   MfgOrders_OrderName : ALIAS FOR WC_L.FlexSTRING[3];
   MfgOrders_PartName : ALIAS FOR WC_L.FlexSTRING[0];
   Motion : DINT := 13;
   Motion1Bit : BOOL := 1;
   Motion_Counter : DINT := 1;
   Motion_Speed : DINT := 12;
   MotionCount : TIMER := (PRE := 1080);
   MotionHolder1 : DINT := 17;
   OEE : OEE := (IdealCycleTime := 3.0);
   OEE_IdealCycleTime : ALIAS FOR WC_L.IdealCT;
   OEE_Parts_Good : ALIAS FOR WC_L.GoodParts;
   OEE_Parts_Scrap : ALIAS FOR WC_L.ScrapParts;
   OEE_Parts_Total : ALIAS FOR WC_L.TotalParts;
   onsbits : DINT;
   OperatorID : ALIAS FOR WC_L.FlexREAL[1];
   Pressure1 : ALIAS FOR WC_L.PV[0];   // PSI
   ProductColorCode : INT := 2;
   Reset1Bit : BOOL;
   SecondTimer : TIMER := (PRE := 60000, ACC := 8545, EN := 1, TT := 1);
   SIM : SimVars := (Run.PRE := 59634, Event.PRE := 4000, Setup.PRE := 4000, EventNumber := 2, UtilityBool[2] := 1);
        .UTILITYBOOL[2]   // First Scan Bit
   Starve_Delay : TIMER := (PRE := 15000);
   Starved_L : BOOL;
   Starved_L1 : BOOL;
   StateValue : ALIAS FOR WC_L.MonitorValue[0];
   Suppress : Events;
   Temperature1 : ALIAS FOR WC_L.PV[1];   // DEG
   UpStream_Run : ALIAS FOR WC[1].EventTrigger[0].1;
   UpStream_Running : ALIAS FOR WC[1].EventTrigger[0].8;
   WC_L : ALIAS FOR WC[3];
END_VAR

ROUTINE MainRoutine   (* ladder *)
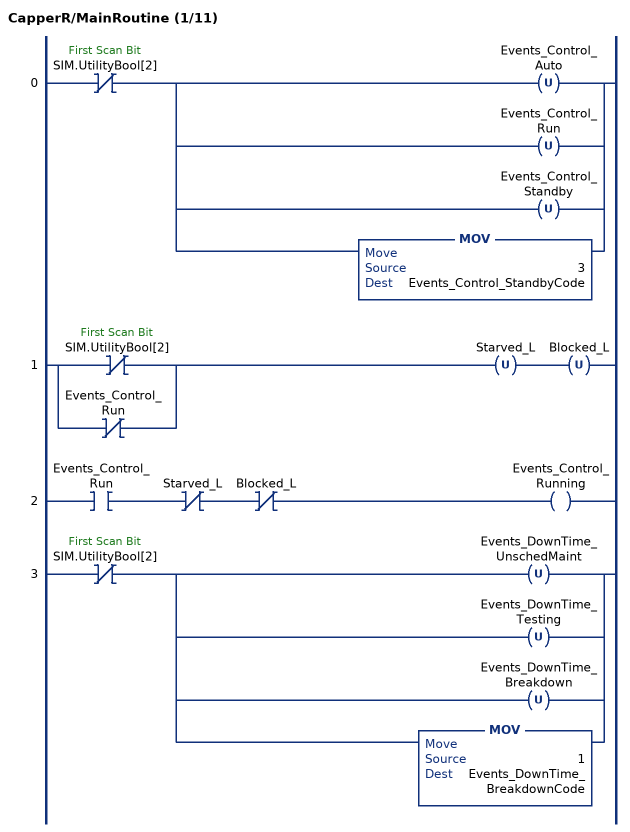
   0: XIO(SIM.UtilityBool[2])[OTU(Events_Control_Auto) ,OTU(Events_Control_Run) ,OTU(Events_Control_Standby) ,MOV(3,Events_Control_StandbyCode) ];
   1: [XIO(SIM.UtilityBool[2]) ,XIO(Events_Control_Run) ]OTU(Starved_L)OTU(Blocked_L);
   2: XIC(Events_Control_Run)XIO(Starved_L)XIO(Blocked_L)OTE(Events_Control_Running);
   3: XIO(SIM.UtilityBool[2])[OTU(Events_DownTime_UnschedMaint) ,OTU(Events_DownTime_Testing) ,OTU(Events_DownTime_Breakdown) ,MOV(1,Events_DownTime_BreakdownCode) ];
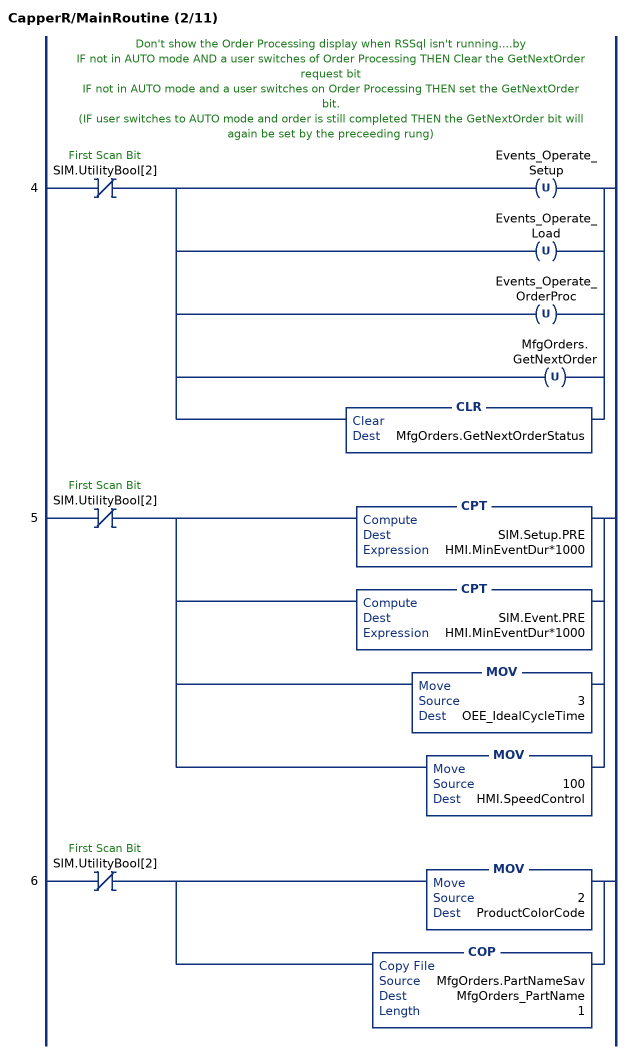
   // Don't show the Order Processing display when RSSql isn't running....by
   // IF not in AUTO mode AND a user switches of Order Processing THEN Clear the GetNextOrder request bit
   // IF not in AUTO mode and a user switches on Order Processing THEN set the GetNextOrder bit.
   // (IF user switches to AUTO mode and order is still completed THEN the GetNextOrder bit will again be set by the preceeding rung)
   4: XIO(SIM.UtilityBool[2])[OTU(Events_Operate_Setup) ,OTU(Events_Operate_Load) ,OTU(Events_Operate_OrderProc) ,OTU(MfgOrders.GetNextOrder) ,CLR(MfgOrders.GetNextOrderStatus) ];
   5: XIO(SIM.UtilityBool[2])[CPT(SIM.Setup.PRE,HMI.MinEventDur*1000) ,CPT(SIM.Event.PRE,HMI.MinEventDur*1000) ,MOV(3,OEE_IdealCycleTime) ,MOV(100,HMI.SpeedControl) ];
   6: XIO(SIM.UtilityBool[2])[MOV(2,ProductColorCode) ,COP(MfgOrders.PartNameSav,MfgOrders_PartName,1) ];
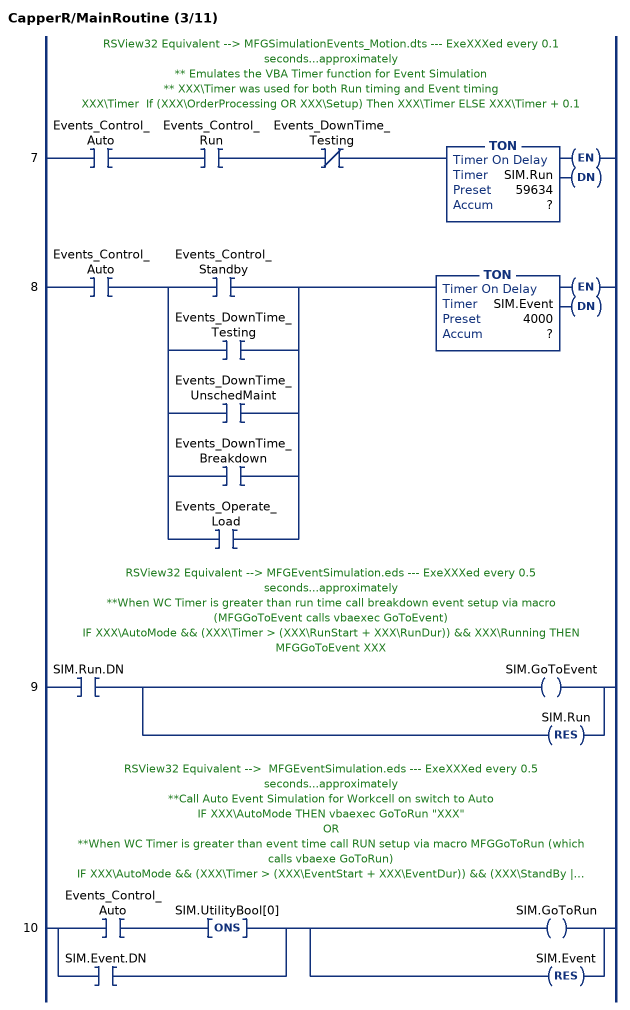
   // RSView32 Equivalent --> MFGSimulationEvents_Motion.dts --- ExeXXXed every 0.1 seconds...approximately
   // ** Emulates the VBA Timer function for Event Simulation
   // ** XXX\Timer was used for both Run timing and Event timing
   // XXX\Timer	If (XXX\OrderProcessing OR XXX\Setup) Then XXX\Timer ELSE XXX\Timer + 0.1
   7: XIC(Events_Control_Auto)XIC(Events_Control_Run)XIO(Events_DownTime_Testing)TON(SIM.Run,?,?);
   8: XIC(Events_Control_Auto)[XIC(Events_Control_Standby) ,XIC(Events_DownTime_Testing) ,XIC(Events_DownTime_UnschedMaint) ,XIC(Events_DownTime_Breakdown) ,XIC(Events_Operate_Load) ]TON(SIM.Event,?,?);
   // RSView32 Equivalent --> MFGEventSimulation.eds --- ExeXXXed every 0.5 seconds...approximately
   // **When WC Timer is greater than run time call breakdown event setup via macro (MFGGoToEvent calls vbaexec GoToEvent)
   // IF XXX\AutoMode && (XXX\Timer > (XXX\RunStart + XXX\RunDur)) && XXX\Running THEN MFGGoToEvent XXX
   9: XIC(SIM.Run.DN)[OTE(SIM.GoToEvent) ,RES(SIM.Run) ];
   // RSView32 Equivalent -->  MFGEventSimulation.eds --- ExeXXXed every 0.5 seconds...approximately
   // **Call Auto Event Simulation for Workcell on switch to Auto
   // IF XXX\AutoMode THEN vbaexec GoToRun "XXX"
   // OR
   // **When WC Timer is greater than event time call RUN setup via macro MFGGoToRun (which calls vbaexe GoToRun)
   // IF XXX\AutoMode && (XXX\Timer > (XXX\EventStart + XXX\EventDur)) && (XXX\StandBy || XXX\Test || XXX\UnSchedMaint || XXX\Breakdown ||XXX\Load) THEN MFGGoToRun XXX
   10: [XIC(Events_Control_Auto) ONS(SIM.UtilityBool[0]) ,XIC(SIM.Event.DN) ][OTE(SIM.GoToRun) ,RES(SIM.Event) ];
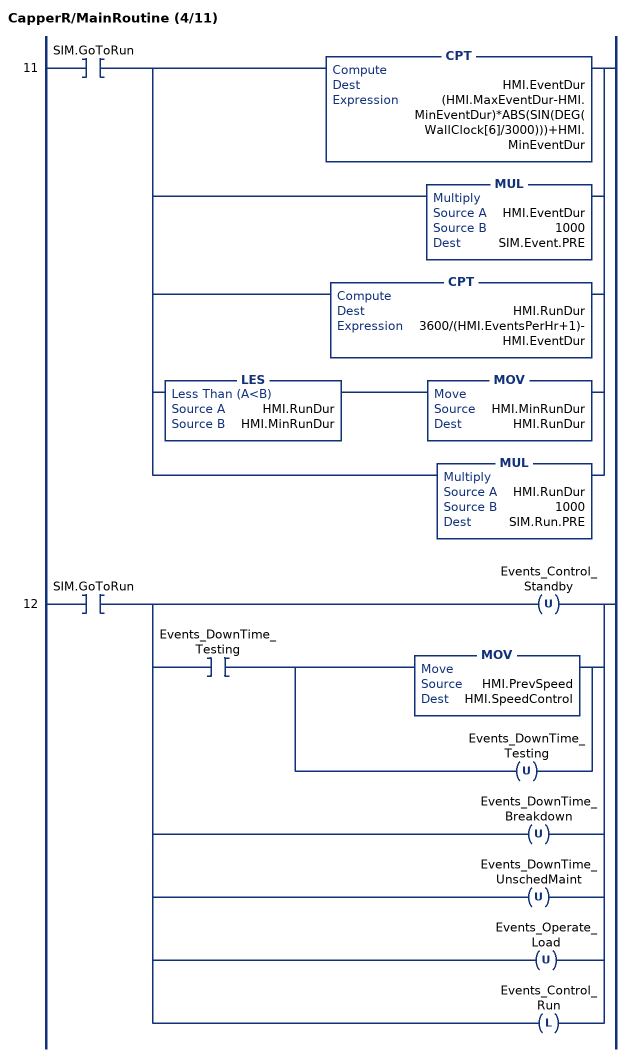
   11: XIC(SIM.GoToRun)[CPT(HMI.EventDur,(HMI.MaxEventDur-HMI.MinEventDur)*ABS(SIN(DEG(WallClock[6]/3000)))+HMI.MinEventDur) ,MUL(HMI.EventDur,1000,SIM.Event.PRE) ,CPT(HMI.RunDur,3600/(HMI.EventsPerHr+1)-HMI.EventDur) ,LES(HMI.RunDur,HMI.MinRunDur) MOV(HMI.MinRunDur,HMI.RunDur) ,MUL(HMI.RunDur,1000,SIM.Run.PRE) ];
   12: XIC(SIM.GoToRun)[OTU(Events_Control_Standby) ,XIC(Events_DownTime_Testing) [MOV(HMI.PrevSpeed,HMI.SpeedControl) ,OTU(Events_DownTime_Testing) ] ,OTU(Events_DownTime_Breakdown) ,OTU(Events_DownTime_UnschedMaint) ,OTU(Events_Operate_Load) ,OTL(Events_Control_Run) ];
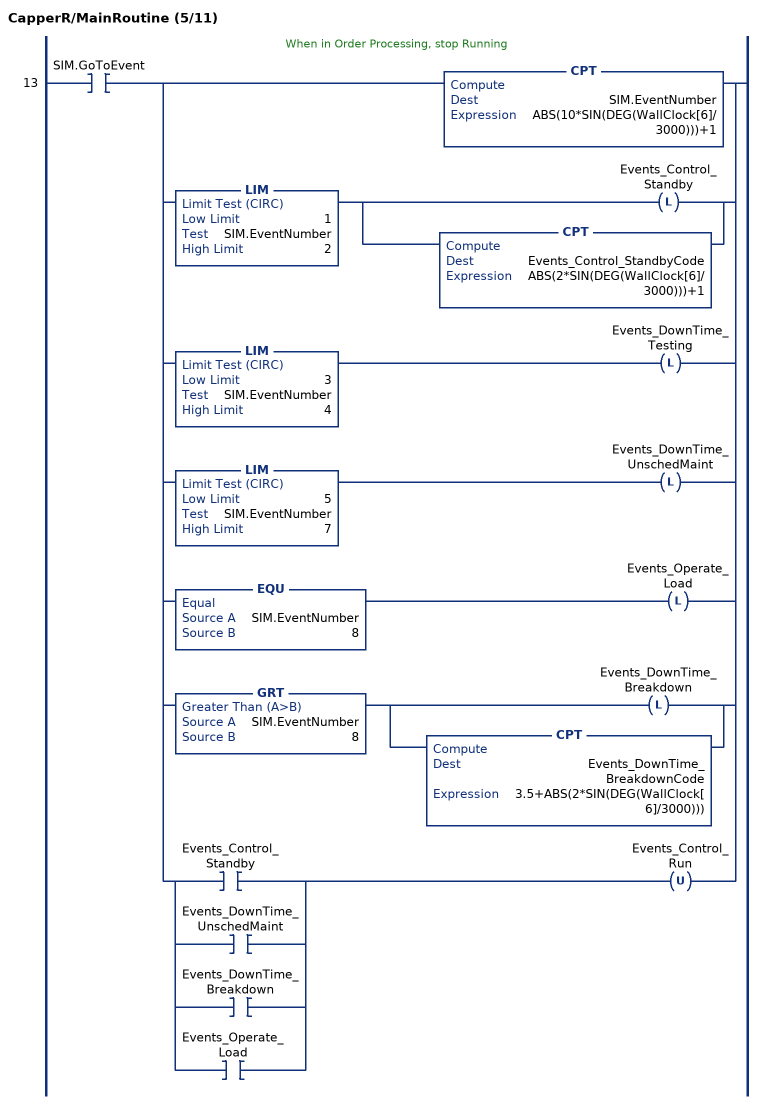
   // When in Order Processing, stop Running
   13: XIC(SIM.GoToEvent)[CPT(SIM.EventNumber,ABS(10*SIN(DEG(WallClock[6]/3000)))+1) ,LIM(1,SIM.EventNumber,2) [OTL(Events_Control_Standby) ,CPT(Events_Control_StandbyCode,ABS(2*SIN(DEG(WallClock[6]/3000)))+1) ] ,LIM(3,SIM.EventNumber,4) OTL(Events_DownTime_Testing) ,LIM(5,SIM.EventNumber,7) OTL(Events_DownTime_UnschedMaint) ,EQU(SIM.EventNumber,8) OTL(Events_Operate_Load) ,GRT(SIM.EventNumber,8) [OTL(Events_DownTime_Breakdown) ,CPT(Events_DownTime_BreakdownCode,3.5+ABS(2*SIN(DEG(WallClock[6]/3000)))) ] ,[XIC(Events_Control_Standby) ,XIC(Events_DownTime_UnschedMaint) ,XIC(Events_DownTime_Breakdown) ,XIC(Events_Operate_Load) ] OTU(Events_Control_Run) ];
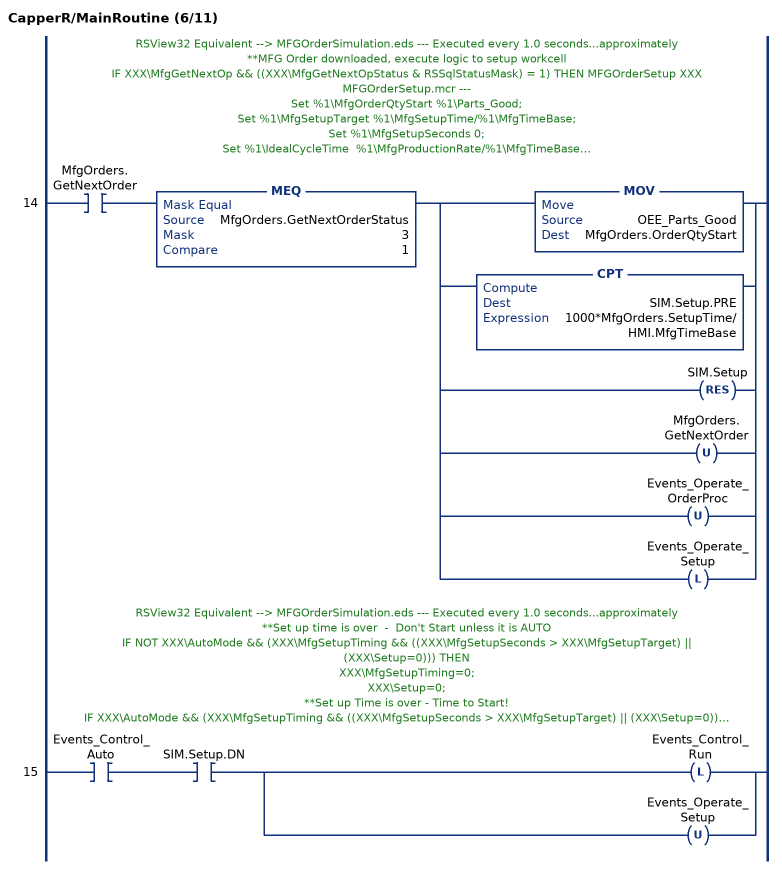
   // RSView32 Equivalent --> MFGOrderSimulation.eds --- Executed every 1.0 seconds...approximately
   // **MFG Order downloaded, execute logic to setup workcell
   // IF XXX\MfgGetNextOp && ((XXX\MfgGetNextOpStatus & RSSqlStatusMask) = 1) THEN MFGOrderSetup XXX
   // MFGOrderSetup.mcr ---
   // 	Set %1\MfgOrderQtyStart %1\Parts_Good;
   // 	Set %1\MfgSetupTarget %1\MfgSetupTime/%1\MfgTimeBase;
   // 	Set %1\MfgSetupSeconds 0;
   // 	Set %1\IdealCycleTime  %1\MfgProductionRate/%1\MfgTimeBase;
   // 	Set %1\MfgGetNextOp 0;
   // 	Set %1\Setup 1;
   // 	Set %1\OrderProcessing 0;
   // 	Set %1\MfgSetupTiming 1;
   14: XIC(MfgOrders.GetNextOrder)MEQ(MfgOrders.GetNextOrderStatus,3,1)[MOV(OEE_Parts_Good,MfgOrders.OrderQtyStart) ,CPT(SIM.Setup.PRE,1000*MfgOrders.SetupTime/HMI.MfgTimeBase) ,RES(SIM.Setup) ,OTU(MfgOrders.GetNextOrder) ,OTU(Events_Operate_OrderProc) ,OTL(Events_Operate_Setup) ];
   // RSView32 Equivalent --> MFGOrderSimulation.eds --- Executed every 1.0 seconds...approximately
   // **Set up time is over  -  Don't Start unless it is AUTO
   // IF NOT XXX\AutoMode && (XXX\MfgSetupTiming && ((XXX\MfgSetupSeconds > XXX\MfgSetupTarget) || (XXX\Setup=0))) THEN
   // 	XXX\MfgSetupTiming=0;
   // 	XXX\Setup=0;
   // **Set up Time is over - Time to Start!
   // IF XXX\AutoMode && (XXX\MfgSetupTiming && ((XXX\MfgSetupSeconds > XXX\MfgSetupTarget) || (XXX\Setup=0))) THEN
   // 	XXX\MfgSetupTiming=0;
   // 	XXX\Setup=0;
   // 	XXX\RUNNING=1
   15: XIC(Events_Control_Auto)XIC(SIM.Setup.DN)[OTL(Events_Control_Run) ,OTU(Events_Operate_Setup) ];
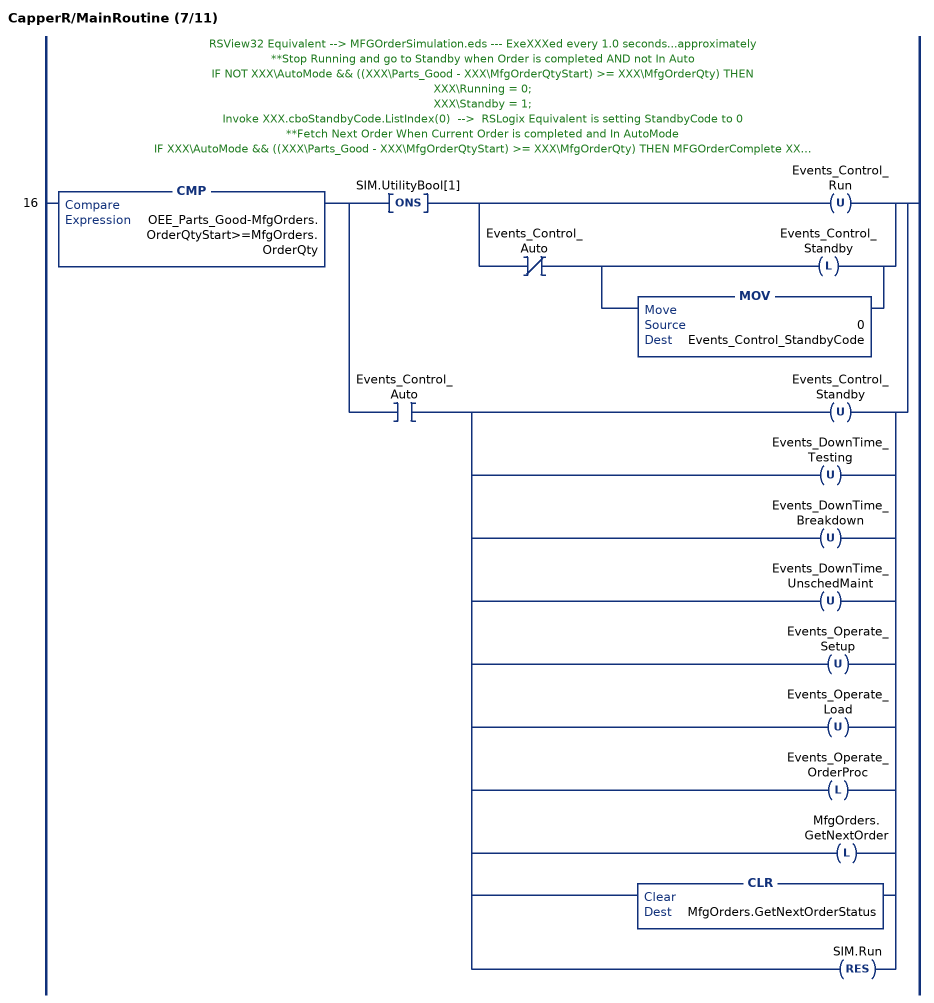
   // RSView32 Equivalent --> MFGOrderSimulation.eds --- ExeXXXed every 1.0 seconds...approximately
   // **Stop Running and go to Standby when Order is completed AND not In Auto
   // IF NOT XXX\AutoMode && ((XXX\Parts_Good - XXX\MfgOrderQtyStart) >= XXX\MfgOrderQty) THEN
   // 	XXX\Running = 0;
   // 	XXX\Standby = 1;
   // 	Invoke XXX.cboStandbyCode.ListIndex(0)  -->  RSLogix Equivalent is setting StandbyCode to 0
   // **Fetch Next Order When Current Order is completed and In AutoMode
   // IF XXX\AutoMode && ((XXX\Parts_Good - XXX\MfgOrderQtyStart) >= XXX\MfgOrderQty) THEN MFGOrderComplete XXX
   // MFGOrderComplete.mcr --- (Macros exeXXXed when called. %1 is the Workcell name -- typical all mcrs)
   // 	Set %1\RunStart %1\Timer;
   // 	Set %1\StandBy 0;
   // 	Set %1\Test 0;
   // 	Set %1\UnSchedMaint 0;
   // 	Set %1\Breakdown 0;
   // 	Set %1\Load 0;
   // 	Set %1\OrderProcessing 1;
   // 	Set %1\Running 0;
   // 	Set %1\MFGGetNextOpStatus 0;
   // 	Set %1\MFGGetNextOp 1
   16: CMP(OEE_Parts_Good-MfgOrders.OrderQtyStart>=MfgOrders.OrderQty)[ONS(SIM.UtilityBool[1]) [OTU(Events_Control_Run) ,XIO(Events_Control_Auto) [OTL(Events_Control_Standby) ,MOV(0,Events_Control_StandbyCode) ] ] ,XIC(Events_Control_Auto) [OTU(Events_Control_Standby) ,OTU(Events_DownTime_Testing) ,OTU(Events_DownTime_Breakdown) ,OTU(Events_DownTime_UnschedMaint) ,OTU(Events_Operate_Setup) ,OTU(Events_Operate_Load) ,OTL(Events_Operate_OrderProc) ,OTL(MfgOrders.GetNextOrder) ,CLR(MfgOrders.GetNextOrderStatus) ,RES(SIM.Run) ] ];
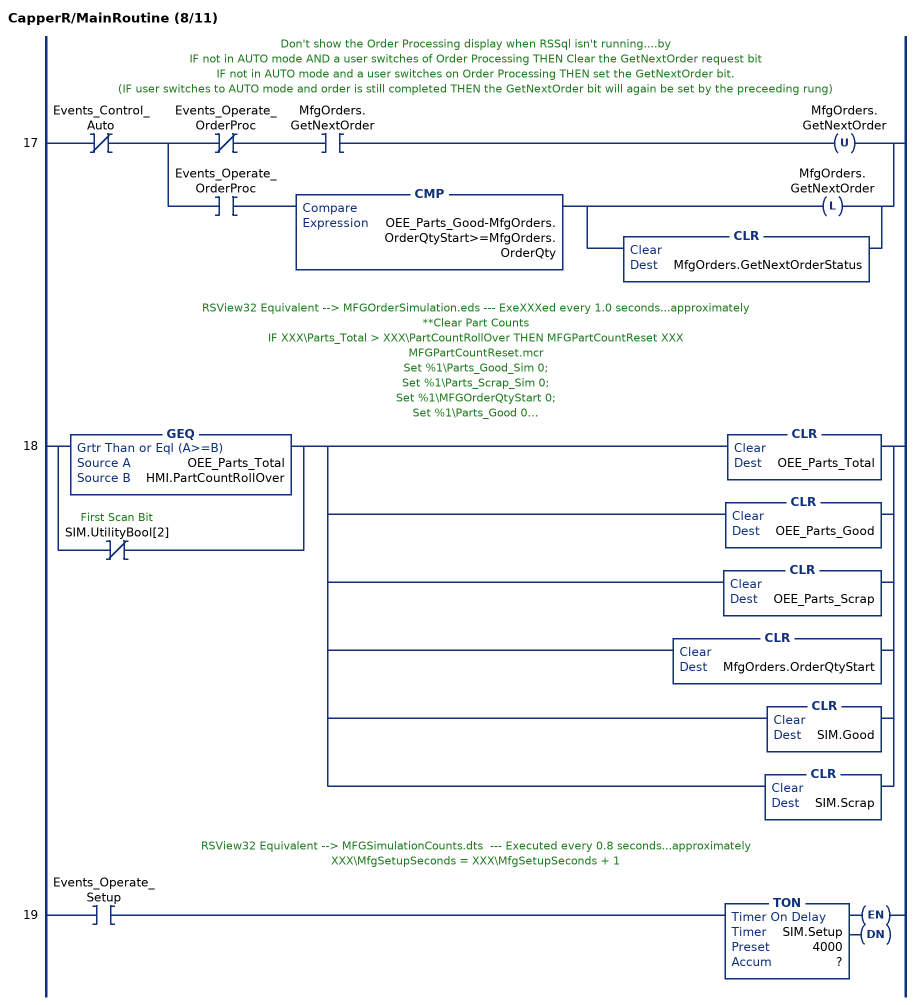
   // Don't show the Order Processing display when RSSql isn't running....by
   // IF not in AUTO mode AND a user switches of Order Processing THEN Clear the GetNextOrder request bit
   // IF not in AUTO mode and a user switches on Order Processing THEN set the GetNextOrder bit.
   // (IF user switches to AUTO mode and order is still completed THEN the GetNextOrder bit will again be set by the preceeding rung)
   17: XIO(Events_Control_Auto)[XIO(Events_Operate_OrderProc) XIC(MfgOrders.GetNextOrder) OTU(MfgOrders.GetNextOrder) ,XIC(Events_Operate_OrderProc) CMP(OEE_Parts_Good-MfgOrders.OrderQtyStart>=MfgOrders.OrderQty) [OTL(MfgOrders.GetNextOrder) ,CLR(MfgOrders.GetNextOrderStatus) ] ];
   // RSView32 Equivalent --> MFGOrderSimulation.eds --- ExeXXXed every 1.0 seconds...approximately
   // **Clear Part Counts
   // IF XXX\Parts_Total > XXX\PartCountRollOver THEN MFGPartCountReset XXX
   // MFGPartCountReset.mcr
   // 	Set %1\Parts_Good_Sim 0;
   // 	Set %1\Parts_Scrap_Sim 0;
   // 	Set %1\MFGOrderQtyStart 0;
   // 	Set %1\Parts_Good 0;
   // 	Set %1\Parts_Scrap 0;
   // 	Set %1\Parts_Total 0
   18: [GEQ(OEE_Parts_Total,HMI.PartCountRollOver) ,XIO(SIM.UtilityBool[2]) ][CLR(OEE_Parts_Total) ,CLR(OEE_Parts_Good) ,CLR(OEE_Parts_Scrap) ,CLR(MfgOrders.OrderQtyStart) ,CLR(SIM.Good) ,CLR(SIM.Scrap) ];
   // RSView32 Equivalent --> MFGSimulationCounts.dts	--- Executed every 0.8 seconds...approximately
   // XXX\MfgSetupSeconds = XXX\MfgSetupSeconds + 1
   19: XIC(Events_Operate_Setup)TON(SIM.Setup,?,?);
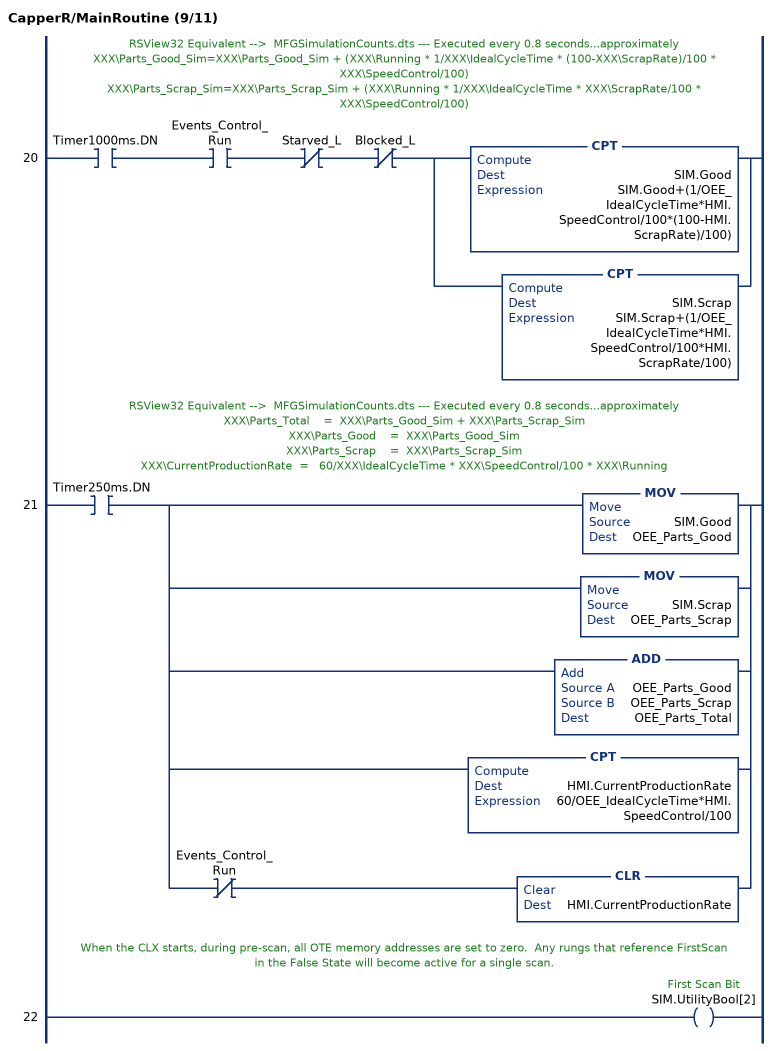
   // RSView32 Equivalent -->  MFGSimulationCounts.dts --- Executed every 0.8 seconds...approximately
   // XXX\Parts_Good_Sim=XXX\Parts_Good_Sim + (XXX\Running * 1/XXX\IdealCycleTime * (100-XXX\ScrapRate)/100 * XXX\SpeedControl/100)
   // XXX\Parts_Scrap_Sim=XXX\Parts_Scrap_Sim + (XXX\Running * 1/XXX\IdealCycleTime * XXX\ScrapRate/100 * XXX\SpeedControl/100)
   20: XIC(Timer1000ms.DN)XIC(Events_Control_Run)XIO(Starved_L)XIO(Blocked_L)[CPT(SIM.Good,SIM.Good+(1/OEE_IdealCycleTime*HMI.SpeedControl/100*(100-HMI.ScrapRate)/100)) ,CPT(SIM.Scrap,SIM.Scrap+(1/OEE_IdealCycleTime*HMI.SpeedControl/100*HMI.ScrapRate/100)) ];
   // RSView32 Equivalent -->  MFGSimulationCounts.dts --- Executed every 0.8 seconds...approximately
   // XXX\Parts_Total		=	XXX\Parts_Good_Sim + XXX\Parts_Scrap_Sim
   // XXX\Parts_Good		=	XXX\Parts_Good_Sim
   // XXX\Parts_Scrap		=	XXX\Parts_Scrap_Sim
   // XXX\CurrentProductionRate  = 	60/XXX\IdealCycleTime * XXX\SpeedControl/100 * XXX\Running
   21: XIC(Timer250ms.DN)[[MOV(SIM.Good,OEE_Parts_Good) ,MOV(SIM.Scrap,OEE_Parts_Scrap) ,ADD(OEE_Parts_Good,OEE_Parts_Scrap,OEE_Parts_Total) ] ,CPT(HMI.CurrentProductionRate,60/OEE_IdealCycleTime*HMI.SpeedControl/100) ,XIO(Events_Control_Run) CLR(HMI.CurrentProductionRate) ];
   // When the CLX starts, during pre-scan, all OTE memory addresses are set to zero.  Any rungs that reference FirstScan in the False State will become active for a single scan.
   22: OTE(SIM.UtilityBool[2]);
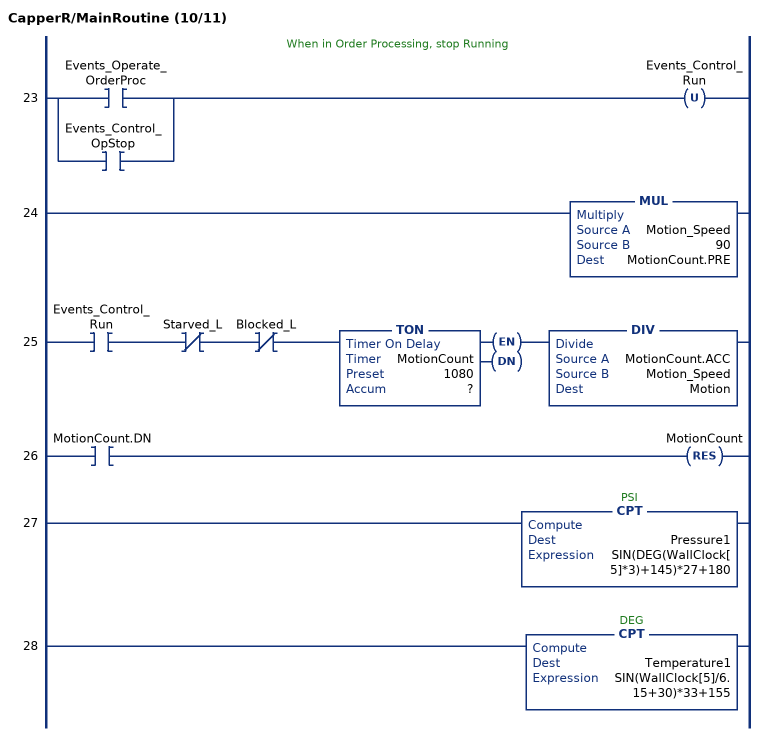
   // When in Order Processing, stop Running
   23: [XIC(Events_Operate_OrderProc) ,XIC(Events_Control_OpStop) ]OTU(Events_Control_Run);
   24: MUL(Motion_Speed,90,MotionCount.PRE);
   25: XIC(Events_Control_Run)XIO(Starved_L)XIO(Blocked_L)TON(MotionCount,?,?)DIV(MotionCount.ACC,Motion_Speed,Motion);
   26: XIC(MotionCount.DN)RES(MotionCount);
   27: CPT(Pressure1,SIN(DEG(WallClock[5]*3)+145)*27+180);
   28: CPT(Temperature1,SIN(WallClock[5]/6.15+30)*33+155);
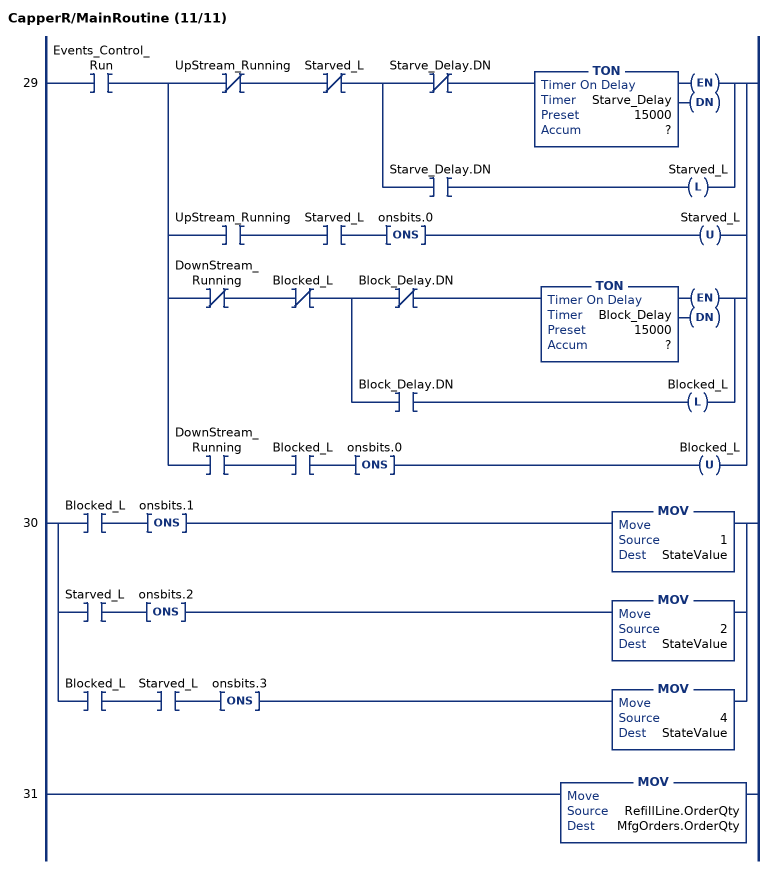
   29: XIC(Events_Control_Run)[[XIO(UpStream_Running) XIO(Starved_L) [XIO(Starve_Delay.DN) TON(Starve_Delay,?,?) ,XIC(Starve_Delay.DN) OTL(Starved_L) ] ,XIC(UpStream_Running) XIC(Starved_L) ONS(onsbits.0) OTU(Starved_L) ] ,[XIO(DownStream_Running) XIO(Blocked_L) [XIO(Block_Delay.DN) TON(Block_Delay,?,?) ,XIC(Block_Delay.DN) OTL(Blocked_L) ] ,XIC(DownStream_Running) XIC(Blocked_L) ONS(onsbits.0) OTU(Blocked_L) ] ];
   30: [XIC(Blocked_L) ONS(onsbits.1) MOV(1,StateValue) ,XIC(Starved_L) ONS(onsbits.2) MOV(2,StateValue) ,XIC(Blocked_L) XIC(Starved_L) ONS(onsbits.3) MOV(4,StateValue) ];
   31: MOV(RefillLine.OrderQty,MfgOrders.OrderQty);
END_ROUTINE
END_PROGRAM
